LIN {X 0,Y 361.85,Z 263.036,A -85,B 0,C 180,E1 -12994.281,E2 -12994.281} C_VEL
LIN {X 0,Y 361.86,Z 263.015,A -85,B 0,C 180,E1 -12997.224,E2 -12997.224} C_VEL
LIN {X 0,Y 361.831,Z 263.036,A -85,B 0,C 180,E1 -13000.756,E2 -13000.756} C_VEL
LIN {X 0,Y 361.816,Z 263.041,A -85,B 0,C 180,E1 -13004.368,E2 -13004.368} C_VEL
LIN {X 0,Y 361.832,Z 262.994,A -85,B 0,C 180,E1 -13007.569,E2 -13007.569} C_VEL
LIN {X 0,Y 361.867,Z 263.034,A -85,B 0,C 180,E1 -13010.974,E2 -13010.974} C_VEL
LIN {X 0,Y 361.871,Z 263.004,A -85,B 0,C 180,E1 -13014.656,E2 -13014.656} C_VEL
LIN {X 0,Y 361.873,Z 263.221,A -85,B 0,C 180,E1 -13016.677,E2 -13016.677} C_VEL
LIN {X 0,Y 365.192,Z 275.83,A -85,B 0,C 180,E1 -13019.658,E2 -13019.658} C_VEL
LIN {X 0,Y 368.197,Z 288.508,A -85,B 0,C 180,E1 -13022.471,E2 -13022.471} C_VEL
LIN {X 0,Y 369.094,Z 293.338,A -85,B 0,C 180,E1 -13023.5,E2 -13023.5} C_VEL
LIN {X 0,Y 368.469,Z 298.908,A -85,B 0,C 180,E1 -13024.51,E2 -13024.51} C_VEL
LIN {X 0,Y 372.505,Z 325.5,A -85,B 0,C 180,E1 -13025.374,E2 -13025.374} C_VEL
LIN {X 0,Y 370.326,Z 430.343,A -85,B 0,C 180,E1 -13027.51,E2 -13027.51} C_VEL
LIN {X 0,Y 369.606,Z 444.397,A -85,B 0,C 180,E1 -13027.979,E2 -13027.979} C_VEL
LIN {X 0,Y 368.698,Z 458.571,A -85,B 0,C 180,E1 -13028.694,E2 -13028.694} C_VEL
LIN {X 0,Y 367.725,Z 471.328,A -85,B 0,C 180,E1 -13029.558,E2 -13029.558} C_VEL
LIN {X 0,Y 366.493,Z 484.339,A -85,B 0,C 180,E1 -13030.684,E2 -13030.684} C_VEL
LIN {X 0,Y 365.21,Z 495.855,A -85,B 0,C 180,E1 -13031.923,E2 -13031.923} C_VEL
LIN {X 0,Y 363.937,Z 507.367,A -85,B 0,C 180,E1 -13033.451,E2 -13033.451} C_VEL
LIN {X 0,Y 362.894,Z 517.59,A -85,B 0,C 180,E1 -13035.132,E2 -13035.132} C_VEL
LIN {X 0,Y 362.087,Z 526.041,A -85,B 0,C 180,E1 -13036.817,E2 -13036.817} C_VEL
LIN {X 0,Y 361.259,Z 534.081,A -85,B 0,C 180,E1 -13038.782,E2 -13038.782} C_VEL
LIN {X 0,Y 360.837,Z 539.679,A -85,B 0,C 180,E1 -13040.471,E2 -13040.471} C_VEL
LIN {X 0,Y 360.561,Z 544.242,A -85,B 0,C 180,E1 -13042.158,E2 -13042.158} C_VEL
LIN {X 0,Y 360.376,Z 548.192,A -85,B 0,C 180,E1 -13044.039,E2 -13044.039} C_VEL
LIN {X 0,Y 360.322,Z 550.495,A -85,B 0,C 180,E1 -13045.525,E2 -13045.525} C_VEL
LIN {X 0,Y 360.262,Z 552.787,A -85,B 0,C 180,E1 -13047.764,E2 -13047.764} C_VEL
LIN {X 0,Y 360.358,Z 553.65,A -85,B 0,C 180,E1 -13050,E2 -13050} C_VEL
LIN {X 0,Y 360.26,Z 553.086,A -85,B 0,C 180,E1 -13052.236,E2 -13052.236} C_VEL
LIN {X 0,Y 360.329,Z 551.079,A -85,B 0,C 180,E1 -13054.475,E2 -13054.475} C_VEL
LIN {X 0,Y 360.479,Z 547.581,A -85,B 0,C 180,E1 -13056.718,E2 -13056.718} C_VEL
LIN {X 0,Y 360.763,Z 542.513,A -85,B 0,C 180,E1 -13058.966,E2 -13058.966} C_VEL
LIN {X 0,Y 361.161,Z 537.589,A -85,B 0,C 180,E1 -13060.653,E2 -13060.653} C_VEL
LIN {X 0,Y 361.961,Z 530.449,A -85,B 0,C 180,E1 -13062.617,E2 -13062.617} C_VEL
LIN {X 0,Y 362.829,Z 522.364,A -85,B 0,C 180,E1 -13064.419,E2 -13064.419} C_VEL
LIN {X 0,Y 363.782,Z 513.901,A -85,B 0,C 180,E1 -13065.98,E2 -13065.98} C_VEL
LIN {X 0,Y 365.146,Z 502.912,A -85,B 0,C 180,E1 -13067.646,E2 -13067.646} C_VEL
LIN {X 0,Y 366.48,Z 491.723,A -85,B 0,C 180,E1 -13069.026,E2 -13069.026} C_VEL
LIN {X 0,Y 367.904,Z 479.321,A -85,B 0,C 180,E1 -13070.255,E2 -13070.255} C_VEL
LIN {X 0,Y 368.921,Z 468.55,A -85,B 0,C 180,E1 -13071.126,E2 -13071.126} C_VEL
LIN {X 0,Y 370.017,Z 455.357,A -85,B 0,C 180,E1 -13071.958,E2 -13071.958} C_VEL
LIN {X 0,Y 370.863,Z 442.406,A -85,B 0,C 180,E1 -13072.566,E2 -13072.566} C_VEL
LIN {X 0,Y 371.556,Z 428.554,A -85,B 0,C 180,E1 -13072.999,E2 -13072.999} C_VEL
LIN {X 0,Y 373.814,Z 326.139,A -85,B 0,C 180,E1 -13075.086,E2 -13075.086} C_VEL
LIN {X 0,Y 369.32,Z 299.055,A -85,B 0,C 180,E1 -13076.023,E2 -13076.023} C_VEL
LIN {X 0,Y 369.764,Z 294.707,A -85,B 0,C 180,E1 -13076.812,E2 -13076.812} C_VEL
LIN {X 0,Y 367.763,Z 285.49,A -85,B 0,C 180,E1 -13078.85,E2 -13078.85} C_VEL
LIN {X 0,Y 364.404,Z 272.229,A -85,B 0,C 180,E1 -13081.941,E2 -13081.941} C_VEL
LIN {X 0,Y 361.899,Z 263.126,A -85,B 0,C 180,E1 -13084.246,E2 -13084.246} C_VEL
LIN {X 0,Y 361.861,Z 263.004,A -85,B 0,C 180,E1 -13087.222,E2 -13087.222} C_VEL
LIN {X 0,Y 361.902,Z 263.021,A -85,B 0,C 180,E1 -13090.768,E2 -13090.768} C_VEL
LIN {X 0,Y 361.908,Z 263.017,A -85,B 0,C 180,E1 -13094.353,E2 -13094.353} C_VEL
LIN {X 0,Y 361.833,Z 263.032,A -85,B 0,C 180,E1 -13097.568,E2 -13097.568} C_VEL
LIN {X 0,Y 361.867,Z 263.034,A -85,B 0,C 180,E1 -13100.973,E2 -13100.973} C_VEL
LIN {X 0,Y 361.87,Z 263.017,A -85,B 0,C 180,E1 -13104.655,E2 -13104.655} C_VEL
LIN {X 0,Y 361.833,Z 263.029,A -85,B 0,C 180,E1 -13108.37,E2 -13108.37} C_VEL
LIN {X 0,Y 361.897,Z 263.009,A -85,B 0,C 180,E1 -13110.955,E2 -13110.955} C_VEL
LIN {X 0,Y 361.95,Z 263.023,A -85,B 0,C 180,E1 -13113.475,E2 -13113.475} C_VEL
LIN {X 0,Y 361.885,Z 263.03,A -85,B 0,C 180,E1 -13117.145,E2 -13117.145} C_VEL
LIN {X 0,Y 361.915,Z 263.026,A -85,B 0,C 180,E1 -13120.724,E2 -13120.724} C_VEL
LIN {X 0,Y 361.94,Z 263.019,A -85,B 0,C 180,E1 -13124.226,E2 -13124.226} C_VEL
LIN {X 0,Y 361.993,Z 263.015,A -85,B 0,C 180,E1 -13126.528,E2 -13126.528} C_VEL
LIN {X 0,Y 362.025,Z 263.016,A -85,B 0,C 180,E1 -13129.938,E2 -13129.938} C_VEL
LIN {X 0,Y 362.157,Z 262.988,A -85,B 0,C 180,E1 -13133.314,E2 -13133.314} C_VEL
LIN {X 0,Y 362.277,Z 262.975,A -85,B 0,C 180,E1 -13137.777,E2 -13137.777} C_VEL
LIN {X 0,Y 362.422,Z 262.965,A -85,B 0,C 180,E1 -13140,E2 -13140} C_VEL
LIN {X 0,Y 362.277,Z 262.972,A -85,B 0,C 180,E1 -13142.224,E2 -13142.224} C_VEL
LIN {X 0,Y 362.166,Z 262.989,A -85,B 0,C 180,E1 -13146.687,E2 -13146.687} C_VEL
LIN {X 0,Y 362.069,Z 263.007,A -85,B 0,C 180,E1 -13148.934,E2 -13148.934} C_VEL
LIN {X 0,Y 361.955,Z 263.017,A -85,B 0,C 180,E1 -13152.333,E2 -13152.333} C_VEL
LIN {X 0,Y 361.957,Z 263.021,A -85,B 0,C 180,E1 -13154.621,E2 -13154.621} C_VEL
LIN {X 0,Y 361.952,Z 263.022,A -85,B 0,C 180,E1 -13158.1,E2 -13158.1} C_VEL
LIN {X 0,Y 361.89,Z 263.032,A -85,B 0,C 180,E1 -13161.654,E2 -13161.654} C_VEL
LIN {X 0,Y 361.925,Z 263.03,A -85,B 0,C 180,E1 -13165.291,E2 -13165.291} C_VEL
LIN {X 0,Y 361.905,Z 263.016,A -85,B 0,C 180,E1 -13167.78,E2 -13167.78} C_VEL
LIN {X 0,Y 361.835,Z 263.039,A -85,B 0,C 180,E1 -13171.63,E2 -13171.63} C_VEL
LIN {X 0,Y 361.873,Z 263.016,A -85,B 0,C 180,E1 -13175.346,E2 -13175.346} C_VEL
LIN {X 0,Y 361.868,Z 263.023,A -85,B 0,C 180,E1 -13179.027,E2 -13179.027} C_VEL
LIN {X 0,Y 361.835,Z 263.035,A -85,B 0,C 180,E1 -13182.83,E2 -13182.83} C_VEL
LIN {X 0,Y 361.82,Z 263.042,A -85,B 0,C 180,E1 -13185.947,E2 -13185.947} C_VEL
LIN {X 0,Y 361.838,Z 263.039,A -85,B 0,C 180,E1 -13189.245,E2 -13189.245} C_VEL
LIN {X 0,Y 361.865,Z 263.007,A -85,B 0,C 180,E1 -13192.778,E2 -13192.778} C_VEL
LIN {X 0,Y 361.888,Z 263.182,A -85,B 0,C 180,E1 -13193.42,E2 -13193.42} C_VEL
LIN {X 0,Y 364.744,Z 273.91,A -85,B 0,C 180,E1 -13196.286,E2 -13196.286} C_VEL
LIN {X 0,Y 367.578,Z 286.235,A -85,B 0,C 180,E1 -13199.361,E2 -13199.361} C_VEL
LIN {X 0,Y 368.84,Z 292.603,A -85,B 0,C 180,E1 -13200.881,E2 -13200.881} C_VEL
LIN {X 0,Y 367.561,Z 304.193,A -85,B 0,C 180,E1 -13203.299,E2 -13203.299} C_VEL
LIN {X 0,Y 366.772,Z 311.792,A -85,B 0,C 180,E1 -13204.83,E2 -13204.83} C_VEL
LIN {X 0,Y 370.593,Z 331.748,A -85,B 0,C 180,E1 -13205.546,E2 -13205.546} C_VEL
LIN {X 0,Y 372.973,Z 345.776,A -85,B 0,C 180,E1 -13205.987,E2 -13205.987} C_VEL
LIN {X 0,Y 371.541,Z 426.495,A -85,B 0,C 180,E1 -13207.478,E2 -13207.478} C_VEL
LIN {X 0,Y 370.858,Z 439.638,A -85,B 0,C 180,E1 -13207.925,E2 -13207.925} C_VEL
LIN {X 0,Y 370.174,Z 451.942,A -85,B 0,C 180,E1 -13208.566,E2 -13208.566} C_VEL
LIN {X 0,Y 369.128,Z 463.623,A -85,B 0,C 180,E1 -13209.377,E2 -13209.377} C_VEL
LIN {X 0,Y 368.017,Z 474.31,A -85,B 0,C 180,E1 -13210.331,E2 -13210.331} C_VEL
LIN {X 0,Y 366.588,Z 485.271,A -85,B 0,C 180,E1 -13211.559,E2 -13211.559} C_VEL
LIN {X 0,Y 365.289,Z 495.077,A -85,B 0,C 180,E1 -13212.938,E2 -13212.938} C_VEL
LIN {X 0,Y 363.91,Z 504.604,A -85,B 0,C 180,E1 -13214.601,E2 -13214.601} C_VEL
LIN {X 0,Y 362.944,Z 512.259,A -85,B 0,C 180,E1 -13216.278,E2 -13216.278} C_VEL
LIN {X 0,Y 362.184,Z 517.473,A -85,B 0,C 180,E1 -13217.676,E2 -13217.676} C_VEL
LIN {X 0,Y 361.451,Z 522.599,A -85,B 0,C 180,E1 -13219.356,E2 -13219.356} C_VEL
LIN {X 0,Y 361.01,Z 526.617,A -85,B 0,C 180,E1 -13221.04,E2 -13221.04} C_VEL
LIN {X 0,Y 360.773,Z 528.765,A -85,B 0,C 180,E1 -13222.163,E2 -13222.163} C_VEL
LIN {X 0,Y 360.453,Z 531.766,A -85,B 0,C 180,E1 -13224.405,E2 -13224.405} C_VEL
LIN {X 0,Y 360.434,Z 532.696,A -85,B 0,C 180,E1 -13225.527,E2 -13225.527} C_VEL
LIN {X 0,Y 360.314,Z 533.479,A -85,B 0,C 180,E1 -13227.764,E2 -13227.764} C_VEL
LIN {X 0,Y 360.365,Z 532.757,A -85,B 0,C 180,E1 -13230,E2 -13230} C_VEL
LIN {X 0,Y 360.523,Z 530.577,A -85,B 0,C 180,E1 -13232.234,E2 -13232.234} C_VEL
LIN {X 0,Y 360.806,Z 527.911,A -85,B 0,C 180,E1 -13233.909,E2 -13233.909} C_VEL
LIN {X 0,Y 361.087,Z 524.308,A -85,B 0,C 180,E1 -13235.585,E2 -13235.585} C_VEL
LIN {X 0,Y 361.638,Z 519.475,A -85,B 0,C 180,E1 -13237.314,E2 -13237.314} C_VEL
LIN {X 0,Y 362.399,Z 512.737,A -85,B 0,C 180,E1 -13239.206,E2 -13239.206} C_VEL
LIN {X 0,Y 363.371,Z 505.272,A -85,B 0,C 180,E1 -13240.869,E2 -13240.869} C_VEL
LIN {X 0,Y 364.513,Z 495.956,A -85,B 0,C 180,E1 -13242.527,E2 -13242.527} C_VEL
LIN {X 0,Y 365.736,Z 485.342,A -85,B 0,C 180,E1 -13244.04,E2 -13244.04} C_VEL
LIN {X 0,Y 366.995,Z 474.475,A -85,B 0,C 180,E1 -13245.266,E2 -13245.266} C_VEL
LIN {X 0,Y 368.083,Z 463.896,A -85,B 0,C 180,E1 -13246.215,E2 -13246.215} C_VEL
LIN {X 0,Y 368.993,Z 452.347,A -85,B 0,C 180,E1 -13247.028,E2 -13247.028} C_VEL
LIN {X 0,Y 369.639,Z 442.84,A -85,B 0,C 180,E1 -13247.543,E2 -13247.543} C_VEL
LIN {X 0,Y 369.41,Z 437.209,A -85,B 0,C 180,E1 -13247.819,E2 -13247.819} C_VEL
LIN {X 0,Y 367.06,Z 428.039,A -85,B 0,C 180,E1 -13248.284,E2 -13248.284} C_VEL
LIN {X 0,Y 364.522,Z 418.753,A -85,B 0,C 180,E1 -13248.664,E2 -13248.664} C_VEL
LIN {X 0,Y 364.025,Z 412.941,A -85,B 0,C 180,E1 -13248.805,E2 -13248.805} C_VEL
LIN {X 0,Y 364.996,Z 345.148,A -85,B 0,C 180,E1 -13250.065,E2 -13250.065} C_VEL
LIN {X 0,Y 359.954,Z 315.672,A -85,B 0,C 180,E1 -13250.989,E2 -13250.989} C_VEL
LIN {X 0,Y 359.295,Z 311.586,A -85,B 0,C 180,E1 -13251.172,E2 -13251.172} C_VEL
LIN {X 0,Y 361.123,Z 294.445,A -85,B 0,C 180,E1 -13254.734,E2 -13254.734} C_VEL
LIN {X 0,Y 361.222,Z 291.662,A -85,B 0,C 180,E1 -13255.342,E2 -13255.342} C_VEL
LIN {X 0,Y 358.66,Z 279.164,A -85,B 0,C 180,E1 -13258.37,E2 -13258.37} C_VEL
LIN {X 0,Y 355.383,Z 266.058,A -85,B 0,C 180,E1 -13261.748,E2 -13261.748} C_VEL
LIN {X 0,Y 354.827,Z 263.972,A -85,B 0,C 180,E1 -13262.371,E2 -13262.371} C_VEL
LIN {X 0,Y 354.823,Z 263.909,A -85,B 0,C 180,E1 -13265.698,E2 -13265.698} C_VEL
LIN {X 0,Y 354.824,Z 263.913,A -85,B 0,C 180,E1 -13269.423,E2 -13269.423} C_VEL
LIN {X 0,Y 354.788,Z 263.917,A -85,B 0,C 180,E1 -13272.866,E2 -13272.866} C_VEL
LIN {X 0,Y 354.766,Z 263.911,A -85,B 0,C 180,E1 -13276.103,E2 -13276.103} C_VEL
LIN {X 0,Y 354.786,Z 263.901,A -85,B 0,C 180,E1 -13279.178,E2 -13279.178} C_VEL
LIN {X 0,Y 354.805,Z 263.911,A -85,B 0,C 180,E1 -13282.402,E2 -13282.402} C_VEL
LIN {X 0,Y 354.809,Z 263.897,A -85,B 0,C 180,E1 -13284.94,E2 -13284.94} C_VEL
LIN {X 0,Y 354.791,Z 263.908,A -85,B 0,C 180,E1 -13288.404,E2 -13288.404} C_VEL
LIN {X 0,Y 354.851,Z 263.9,A -85,B 0,C 180,E1 -13291.618,E2 -13291.618} C_VEL
LIN {X 0,Y 354.895,Z 263.902,A -85,B 0,C 180,E1 -13294.172,E2 -13294.172} C_VEL
LIN {X 0,Y 354.828,Z 263.909,A -85,B 0,C 180,E1 -13297.893,E2 -13297.893} C_VEL
LIN {X 0,Y 354.918,Z 263.897,A -85,B 0,C 180,E1 -13301.891,E2 -13301.891} C_VEL
LIN {X 0,Y 354.937,Z 263.89,A -85,B 0,C 180,E1 -13305.981,E2 -13305.981} C_VEL
LIN {X 0,Y 354.972,Z 263.884,A -85,B 0,C 180,E1 -13309.735,E2 -13309.735} C_VEL
LIN {X 0,Y 355.12,Z 263.873,A -85,B 0,C 180,E1 -13313.18,E2 -13313.18} C_VEL
LIN {X 0,Y 355.24,Z 263.858,A -85,B 0,C 180,E1 -13317.732,E2 -13317.732} C_VEL
LIN {X 0,Y 355.391,Z 263.834,A -85,B 0,C 180,E1 -13320,E2 -13320} C_VEL
LIN {X 0,Y 355.24,Z 263.856,A -85,B 0,C 180,E1 -13322.267,E2 -13322.267} C_VEL
LIN {X 0,Y 355.131,Z 263.868,A -85,B 0,C 180,E1 -13326.819,E2 -13326.819} C_VEL
LIN {X 0,Y 355.009,Z 263.885,A -85,B 0,C 180,E1 -13329.112,E2 -13329.112} C_VEL
LIN {X 0,Y 354.914,Z 263.9,A -85,B 0,C 180,E1 -13332.581,E2 -13332.581} C_VEL
LIN {X 0,Y 354.883,Z 263.896,A -85,B 0,C 180,E1 -13336.096,E2 -13336.096} C_VEL
LIN {X 0,Y 354.897,Z 263.903,A -85,B 0,C 180,E1 -13338.472,E2 -13338.472} C_VEL
LIN {X 0,Y 354.829,Z 263.911,A -85,B 0,C 180,E1 -13342.106,E2 -13342.106} C_VEL
LIN {X 0,Y 354.894,Z 263.899,A -85,B 0,C 180,E1 -13345.828,E2 -13345.828} C_VEL
LIN {X 0,Y 354.849,Z 263.885,A -85,B 0,C 180,E1 -13349.679,E2 -13349.679} C_VEL
LIN {X 0,Y 354.801,Z 263.916,A -85,B 0,C 180,E1 -13353.702,E2 -13353.702} C_VEL
LIN {X 0,Y 354.793,Z 263.895,A -85,B 0,C 180,E1 -13356.46,E2 -13356.46} C_VEL
LIN {X 0,Y 354.819,Z 263.914,A -85,B 0,C 180,E1 -13359.424,E2 -13359.424} C_VEL
LIN {X 0,Y 354.784,Z 263.906,A -85,B 0,C 180,E1 -13362.868,E2 -13362.868} C_VEL
LIN {X 0,Y 354.777,Z 263.898,A -85,B 0,C 180,E1 -13366.106,E2 -13366.106} C_VEL
LIN {X 0,Y 354.783,Z 263.875,A -85,B 0,C 180,E1 -13369.179,E2 -13369.179} C_VEL
LIN {X 0,Y 354.804,Z 263.902,A -85,B 0,C 180,E1 -13372.403,E2 -13372.403} C_VEL
LIN {X 0,Y 354.818,Z 263.969,A -85,B 0,C 180,E1 -13376.07,E2 -13376.07} C_VEL
LIN {X 0,Y 357.55,Z 274.162,A -85,B 0,C 180,E1 -13378.609,E2 -13378.609} C_VEL
LIN {X 0,Y 360.996,Z 288.429,A -85,B 0,C 180,E1 -13381.885,E2 -13381.885} C_VEL
LIN {X 0,Y 362.224,Z 294.363,A -85,B 0,C 180,E1 -13383.19,E2 -13383.19} C_VEL
LIN {X 0,Y 361.79,Z 299.207,A -85,B 0,C 180,E1 -13384.068,E2 -13384.068} C_VEL
LIN {X 0,Y 365.954,Z 326.74,A -85,B 0,C 180,E1 -13384.977,E2 -13384.977} C_VEL
LIN {X 0,Y 363.665,Z 431.378,A -85,B 0,C 180,E1 -13387.15,E2 -13387.15} C_VEL
LIN {X 0,Y 362.85,Z 445.727,A -85,B 0,C 180,E1 -13387.66,E2 -13387.66} C_VEL
LIN {X 0,Y 361.875,Z 459.999,A -85,B 0,C 180,E1 -13388.414,E2 -13388.414} C_VEL
LIN {X 0,Y 360.84,Z 473.26,A -85,B 0,C 180,E1 -13389.361,E2 -13389.361} C_VEL
LIN {X 0,Y 359.604,Z 485.281,A -85,B 0,C 180,E1 -13390.447,E2 -13390.447} C_VEL
LIN {X 0,Y 358.266,Z 496.607,A -85,B 0,C 180,E1 -13391.708,E2 -13391.708} C_VEL
LIN {X 0,Y 357.079,Z 506.996,A -85,B 0,C 180,E1 -13393.124,E2 -13393.124} C_VEL
LIN {X 0,Y 355.968,Z 517.258,A -85,B 0,C 180,E1 -13394.835,E2 -13394.835} C_VEL
LIN {X 0,Y 355.143,Z 525.738,A -85,B 0,C 180,E1 -13396.555,E2 -13396.555} C_VEL
LIN {X 0,Y 354.265,Z 533.801,A -85,B 0,C 180,E1 -13398.558,E2 -13398.558} C_VEL
LIN {X 0,Y 353.787,Z 539.417,A -85,B 0,C 180,E1 -13400.279,E2 -13400.279} C_VEL
LIN {X 0,Y 353.492,Z 543.998,A -85,B 0,C 180,E1 -13402,E2 -13402} C_VEL
LIN {X 0,Y 353.276,Z 548.246,A -85,B 0,C 180,E1 -13404.092,E2 -13404.092} C_VEL
LIN {X 0,Y 353.235,Z 550.272,A -85,B 0,C 180,E1 -13405.435,E2 -13405.435} C_VEL
LIN {X 0,Y 353.17,Z 552.576,A -85,B 0,C 180,E1 -13407.719,E2 -13407.719} C_VEL
LIN {X 0,Y 353.26,Z 553.448,A -85,B 0,C 180,E1 -13410,E2 -13410} C_VEL
LIN {X 0,Y 353.168,Z 552.894,A -85,B 0,C 180,E1 -13412.281,E2 -13412.281} C_VEL
LIN {X 0,Y 353.243,Z 550.899,A -85,B 0,C 180,E1 -13414.565,E2 -13414.565} C_VEL
LIN {X 0,Y 353.388,Z 547.406,A -85,B 0,C 180,E1 -13416.853,E2 -13416.853} C_VEL
LIN {X 0,Y 353.701,Z 542.345,A -85,B 0,C 180,E1 -13419.146,E2 -13419.146} C_VEL
LIN {X 0,Y 354.126,Z 537.425,A -85,B 0,C 180,E1 -13420.867,E2 -13420.867} C_VEL
LIN {X 0,Y 354.983,Z 530.289,A -85,B 0,C 180,E1 -13422.869,E2 -13422.869} C_VEL
LIN {X 0,Y 356.013,Z 521.414,A -85,B 0,C 180,E1 -13424.87,E2 -13424.87} C_VEL
LIN {X 0,Y 357.153,Z 512.096,A -85,B 0,C 180,E1 -13426.578,E2 -13426.578} C_VEL
LIN {X 0,Y 358.481,Z 501.752,A -85,B 0,C 180,E1 -13428.133,E2 -13428.133} C_VEL
LIN {X 0,Y 359.937,Z 490.281,A -85,B 0,C 180,E1 -13429.534,E2 -13429.534} C_VEL
LIN {X 0,Y 361.329,Z 477.518,A -85,B 0,C 180,E1 -13430.794,E2 -13430.794} C_VEL
LIN {X 0,Y 362.584,Z 465.109,A -85,B 0,C 180,E1 -13431.759,E2 -13431.759} C_VEL
LIN {X 0,Y 363.69,Z 451.275,A -85,B 0,C 180,E1 -13432.585,E2 -13432.585} C_VEL
LIN {X 0,Y 364.624,Z 437.641,A -85,B 0,C 180,E1 -13433.161,E2 -13433.161} C_VEL
LIN {X 0,Y 365.152,Z 423.665,A -85,B 0,C 180,E1 -13433.538,E2 -13433.538} C_VEL
LIN {X 0,Y 367.31,Z 326.411,A -85,B 0,C 180,E1 -13435.545,E2 -13435.545} C_VEL
LIN {X 0,Y 362.731,Z 299.025,A -85,B 0,C 180,E1 -13436.535,E2 -13436.535} C_VEL
LIN {X 0,Y 362.956,Z 296.33,A -85,B 0,C 180,E1 -13437.038,E2 -13437.038} C_VEL
LIN {X 0,Y 360.625,Z 285.59,A -85,B 0,C 180,E1 -13439.477,E2 -13439.477} C_VEL
LIN {X 0,Y 357.059,Z 271.925,A -85,B 0,C 180,E1 -13442.77,E2 -13442.77} C_VEL
LIN {X 0,Y 354.844,Z 263.997,A -85,B 0,C 180,E1 -13444.848,E2 -13444.848} C_VEL
LIN {X 0,Y 354.803,Z 263.892,A -85,B 0,C 180,E1 -13447.882,E2 -13447.882} C_VEL
LIN {X 0,Y 354.835,Z 263.901,A -85,B 0,C 180,E1 -13451.18,E2 -13451.18} C_VEL
LIN {X 0,Y 354.859,Z 263.895,A -85,B 0,C 180,E1 -13454.522,E2 -13454.522} C_VEL
LIN {X 0,Y 354.791,Z 263.907,A -85,B 0,C 180,E1 -13457.662,E2 -13457.662} C_VEL
LIN {X 0,Y 354.811,Z 263.914,A -85,B 0,C 180,E1 -13460.666,E2 -13460.666} C_VEL
LIN {X 0,Y 354.818,Z 263.892,A -85,B 0,C 180,E1 -13464.3,E2 -13464.3} C_VEL
LIN {X 0,Y 354.782,Z 263.916,A -85,B 0,C 180,E1 -13467.666,E2 -13467.666} C_VEL
LIN {X 0,Y 354.864,Z 263.881,A -85,B 0,C 180,E1 -13470.621,E2 -13470.621} C_VEL
LIN {X 0,Y 354.894,Z 263.902,A -85,B 0,C 180,E1 -13474.172,E2 -13474.172} C_VEL
LIN {X 0,Y 354.829,Z 263.912,A -85,B 0,C 180,E1 -13477.894,E2 -13477.894} C_VEL
LIN {X 0,Y 354.918,Z 263.901,A -85,B 0,C 180,E1 -13481.891,E2 -13481.891} C_VEL
LIN {X 0,Y 354.937,Z 263.898,A -85,B 0,C 180,E1 -13485.981,E2 -13485.981} C_VEL
LIN {X 0,Y 354.972,Z 263.892,A -85,B 0,C 180,E1 -13489.736,E2 -13489.736} C_VEL
LIN {X 0,Y 355.121,Z 263.863,A -85,B 0,C 180,E1 -13493.181,E2 -13493.181} C_VEL
LIN {X 0,Y 355.24,Z 263.851,A -85,B 0,C 180,E1 -13497.733,E2 -13497.733} C_VEL
LIN {X 0,Y 355.392,Z 263.84,A -85,B 0,C 180,E1 -13500,E2 -13500} C_VEL
LIN {X 0,Y 355.24,Z 263.849,A -85,B 0,C 180,E1 -13502.268,E2 -13502.268} C_VEL
LIN {X 0,Y 355.133,Z 263.864,A -85,B 0,C 180,E1 -13506.82,E2 -13506.82} C_VEL
LIN {X 0,Y 355.01,Z 263.888,A -85,B 0,C 180,E1 -13509.113,E2 -13509.113} C_VEL
LIN {X 0,Y 354.916,Z 263.894,A -85,B 0,C 180,E1 -13512.582,E2 -13512.582} C_VEL
LIN {X 0,Y 354.885,Z 263.896,A -85,B 0,C 180,E1 -13516.097,E2 -13516.097} C_VEL
LIN {X 0,Y 354.897,Z 263.901,A -85,B 0,C 180,E1 -13518.473,E2 -13518.473} C_VEL
LIN {X 0,Y 354.832,Z 263.909,A -85,B 0,C 180,E1 -13522.107,E2 -13522.107} C_VEL
LIN {X 0,Y 354.896,Z 263.902,A -85,B 0,C 180,E1 -13525.828,E2 -13525.828} C_VEL
LIN {X 0,Y 354.815,Z 263.891,A -85,B 0,C 180,E1 -13529.683,E2 -13529.683} C_VEL
LIN {X 0,Y 354.804,Z 263.906,A -85,B 0,C 180,E1 -13533.703,E2 -13533.703} C_VEL
LIN {X 0,Y 354.799,Z 263.906,A -85,B 0,C 180,E1 -13536.46,E2 -13536.46} C_VEL
LIN {X 0,Y 354.823,Z 263.897,A -85,B 0,C 180,E1 -13539.425,E2 -13539.425} C_VEL
LIN {X 0,Y 354.787,Z 263.913,A -85,B 0,C 180,E1 -13542.868,E2 -13542.868} C_VEL
LIN {X 0,Y 354.769,Z 263.921,A -85,B 0,C 180,E1 -13546.105,E2 -13546.105} C_VEL
LIN {X 0,Y 354.79,Z 263.918,A -85,B 0,C 180,E1 -13549.18,E2 -13549.18} C_VEL
LIN {X 0,Y 354.844,Z 264.023,A -85,B 0,C 180,E1 -13552.811,E2 -13552.811} C_VEL
LIN {X 0,Y 357.595,Z 274.245,A -85,B 0,C 180,E1 -13555.635,E2 -13555.635} C_VEL
LIN {X 0,Y 360.671,Z 287.482,A -85,B 0,C 180,E1 -13559.025,E2 -13559.025} C_VEL
LIN {X 0,Y 362.001,Z 294.128,A -85,B 0,C 180,E1 -13560.647,E2 -13560.647} C_VEL
LIN {X 0,Y 361.283,Z 301.246,A -85,B 0,C 180,E1 -13562.169,E2 -13562.169} C_VEL
LIN {X 0,Y 360.095,Z 311.644,A -85,B 0,C 180,E1 -13564.32,E2 -13564.32} C_VEL
LIN {X 0,Y 364.167,Z 332.827,A -85,B 0,C 180,E1 -13565.102,E2 -13565.102} C_VEL
LIN {X 0,Y 366.514,Z 346.606,A -85,B 0,C 180,E1 -13565.548,E2 -13565.548} C_VEL
LIN {X 0,Y 365.011,Z 426.627,A -85,B 0,C 180,E1 -13567.052,E2 -13567.052} C_VEL
LIN {X 0,Y 364.271,Z 439.964,A -85,B 0,C 180,E1 -13567.515,E2 -13567.515} C_VEL
LIN {X 0,Y 363.57,Z 452.04,A -85,B 0,C 180,E1 -13568.157,E2 -13568.157} C_VEL
LIN {X 0,Y 362.495,Z 463.721,A -85,B 0,C 180,E1 -13568.981,E2 -13568.981} C_VEL
LIN {X 0,Y 361.326,Z 474.411,A -85,B 0,C 180,E1 -13569.952,E2 -13569.952} C_VEL
LIN {X 0,Y 359.861,Z 485.379,A -85,B 0,C 180,E1 -13571.202,E2 -13571.202} C_VEL
LIN {X 0,Y 358.474,Z 495.191,A -85,B 0,C 180,E1 -13572.604,E2 -13572.604} C_VEL
LIN {X 0,Y 357.046,Z 504.726,A -85,B 0,C 180,E1 -13574.298,E2 -13574.298} C_VEL
LIN {X 0,Y 356,Z 512.427,A -85,B 0,C 180,E1 -13576.014,E2 -13576.014} C_VEL
LIN {X 0,Y 355.245,Z 517.612,A -85,B 0,C 180,E1 -13577.431,E2 -13577.431} C_VEL
LIN {X 0,Y 354.451,Z 522.747,A -85,B 0,C 180,E1 -13579.143,E2 -13579.143} C_VEL
LIN {X 0,Y 353.96,Z 526.776,A -85,B 0,C 180,E1 -13580.86,E2 -13580.86} C_VEL
LIN {X 0,Y 353.719,Z 528.928,A -85,B 0,C 180,E1 -13582.005,E2 -13582.005} C_VEL
LIN {X 0,Y 353.438,Z 531.496,A -85,B 0,C 180,E1 -13583.851,E2 -13583.851} C_VEL
LIN {X 0,Y 353.344,Z 532.88,A -85,B 0,C 180,E1 -13585.437,E2 -13585.437} C_VEL
LIN {X 0,Y 353.22,Z 533.675,A -85,B 0,C 180,E1 -13587.719,E2 -13587.719} C_VEL
LIN {X 0,Y 353.247,Z 533.512,A -85,B 0,C 180,E1 -13588.86,E2 -13588.86} C_VEL
LIN {X 0,Y 353.323,Z 532.073,A -85,B 0,C 180,E1 -13591.14,E2 -13591.14} C_VEL
LIN {X 0,Y 353.588,Z 529.163,A -85,B 0,C 180,E1 -13593.418,E2 -13593.418} C_VEL
LIN {X 0,Y 353.882,Z 525.888,A -85,B 0,C 180,E1 -13595.127,E2 -13595.127} C_VEL
LIN {X 0,Y 354.413,Z 521.609,A -85,B 0,C 180,E1 -13596.833,E2 -13596.833} C_VEL
LIN {X 0,Y 355.141,Z 515.218,A -85,B 0,C 180,E1 -13598.822,E2 -13598.822} C_VEL
LIN {X 0,Y 356.011,Z 508.264,A -85,B 0,C 180,E1 -13600.521,E2 -13600.521} C_VEL
LIN {X 0,Y 357.204,Z 499.651,A -85,B 0,C 180,E1 -13602.21,E2 -13602.21} C_VEL
LIN {X 0,Y 358.315,Z 490.874,A -85,B 0,C 180,E1 -13603.613,E2 -13603.613} C_VEL
LIN {X 0,Y 359.457,Z 481.27,A -85,B 0,C 180,E1 -13604.869,E2 -13604.869} C_VEL
LIN {X 0,Y 360.584,Z 470.793,A -85,B 0,C 180,E1 -13605.98,E2 -13605.98} C_VEL
LIN {X 0,Y 361.73,Z 459.246,A -85,B 0,C 180,E1 -13606.943,E2 -13606.943} C_VEL
LIN {X 0,Y 362.688,Z 447.317,A -85,B 0,C 180,E1 -13607.697,E2 -13607.697} C_VEL
LIN {X 0,Y 363.383,Z 434.196,A -85,B 0,C 180,E1 -13608.29,E2 -13608.29} C_VEL
LIN {X 0,Y 363.859,Z 420.763,A -85,B 0,C 180,E1 -13608.662,E2 -13608.662} C_VEL
LIN {X 0,Y 364.025,Z 412.941,A -85,B 0,C 180,E1 -13608.805,E2 -13608.805} C_VEL
LIN {X 0,Y 363.616,Z 407.128,A -85,B 0,C 180,E1 -13608.943,E2 -13608.943} C_VEL
LIN {X 0,Y 359.05,Z 390.31,A -85,B 0,C 180,E1 -13609.561,E2 -13609.561} C_VEL
LIN {X 0,Y 358.046,Z 384.566,A -85,B 0,C 180,E1 -13609.74,E2 -13609.74} C_VEL
LIN {X 0,Y 357.93,Z 382.612,A -85,B 0,C 180,E1 -13609.787,E2 -13609.787} C_VEL
LIN {X 0,Y 358.472,Z 346.101,A -85,B 0,C 180,E1 -13610.479,E2 -13610.479} C_VEL
LIN {X 0,Y 352.932,Z 313.976,A -85,B 0,C 180,E1 -13611.52,E2 -13611.52} C_VEL
LIN {X 0,Y 352.566,Z 311.323,A -85,B 0,C 180,E1 -13611.673,E2 -13611.673} C_VEL
LIN {X 0,Y 354.482,Z 294.556,A -85,B 0,C 180,E1 -13615.23,E2 -13615.23} C_VEL
LIN {X 0,Y 352.44,Z 283.633,A -85,B 0,C 180,E1 -13617.9,E2 -13617.9} C_VEL
LIN {X 0,Y 349.685,Z 272.324,A -85,B 0,C 180,E1 -13620.829,E2 -13620.829} C_VEL
LIN {X 0,Y 347.779,Z 264.846,A -85,B 0,C 180,E1 -13622.922,E2 -13622.922} C_VEL
LIN {X 0,Y 347.771,Z 264.794,A -85,B 0,C 180,E1 -13626.064,E2 -13626.064} C_VEL
LIN {X 0,Y 347.753,Z 264.791,A -85,B 0,C 180,E1 -13628.792,E2 -13628.792} C_VEL
LIN {X 0,Y 347.751,Z 264.786,A -85,B 0,C 180,E1 -13631.829,E2 -13631.829} C_VEL
LIN {X 0,Y 347.705,Z 264.784,A -85,B 0,C 180,E1 -13635.026,E2 -13635.026} C_VEL
LIN {X 0,Y 347.749,Z 264.791,A -85,B 0,C 180,E1 -13638.396,E2 -13638.396} C_VEL
LIN {X 0,Y 347.772,Z 264.787,A -85,B 0,C 180,E1 -13642.01,E2 -13642.01} C_VEL
LIN {X 0,Y 347.742,Z 264.77,A -85,B 0,C 180,E1 -13645.535,E2 -13645.535} C_VEL
LIN {X 0,Y 347.761,Z 264.791,A -85,B 0,C 180,E1 -13649.653,E2 -13649.653} C_VEL
LIN {X 0,Y 347.849,Z 264.776,A -85,B 0,C 180,E1 -13652.744,E2 -13652.744} C_VEL
LIN {X 0,Y 347.782,Z 264.778,A -85,B 0,C 180,E1 -13656.161,E2 -13656.161} C_VEL
LIN {X 0,Y 347.808,Z 264.778,A -85,B 0,C 180,E1 -13659.909,E2 -13659.909} C_VEL
LIN {X 0,Y 347.861,Z 264.778,A -85,B 0,C 180,E1 -13662.359,E2 -13662.359} C_VEL
LIN {X 0,Y 347.893,Z 264.767,A -85,B 0,C 180,E1 -13665.97,E2 -13665.97} C_VEL
LIN {X 0,Y 347.923,Z 264.762,A -85,B 0,C 180,E1 -13669.525,E2 -13669.525} C_VEL
LIN {X 0,Y 348.086,Z 264.75,A -85,B 0,C 180,E1 -13673.042,E2 -13673.042} C_VEL
LIN {X 0,Y 348.202,Z 264.734,A -85,B 0,C 180,E1 -13677.686,E2 -13677.686} C_VEL
LIN {X 0,Y 348.34,Z 264.712,A -85,B 0,C 180,E1 -13680,E2 -13680} C_VEL
LIN {X 0,Y 348.202,Z 264.733,A -85,B 0,C 180,E1 -13682.313,E2 -13682.313} C_VEL
LIN {X 0,Y 348.1,Z 264.745,A -85,B 0,C 180,E1 -13686.957,E2 -13686.957} C_VEL
LIN {X 0,Y 347.961,Z 264.763,A -85,B 0,C 180,E1 -13689.298,E2 -13689.298} C_VEL
LIN {X 0,Y 347.883,Z 264.775,A -85,B 0,C 180,E1 -13692.839,E2 -13692.839} C_VEL
LIN {X 0,Y 347.833,Z 264.775,A -85,B 0,C 180,E1 -13696.431,E2 -13696.431} C_VEL
LIN {X 0,Y 347.847,Z 264.778,A -85,B 0,C 180,E1 -13698.86,E2 -13698.86} C_VEL
LIN {X 0,Y 347.768,Z 264.791,A -85,B 0,C 180,E1 -13702.579,E2 -13702.579} C_VEL
LIN {X 0,Y 347.806,Z 264.778,A -85,B 0,C 180,E1 -13705.109,E2 -13705.109} C_VEL
LIN {X 0,Y 347.807,Z 264.785,A -85,B 0,C 180,E1 -13707.694,E2 -13707.694} C_VEL
LIN {X 0,Y 347.759,Z 264.764,A -85,B 0,C 180,E1 -13710.347,E2 -13710.347} C_VEL
LIN {X 0,Y 347.74,Z 264.793,A -85,B 0,C 180,E1 -13714.464,E2 -13714.464} C_VEL
LIN {X 0,Y 347.77,Z 264.777,A -85,B 0,C 180,E1 -13717.989,E2 -13717.989} C_VEL
LIN {X 0,Y 347.746,Z 264.779,A -85,B 0,C 180,E1 -13721.831,E2 -13721.831} C_VEL
LIN {X 0,Y 347.762,Z 264.79,A -85,B 0,C 180,E1 -13725.017,E2 -13725.017} C_VEL
LIN {X 0,Y 347.746,Z 264.744,A -85,B 0,C 180,E1 -13728.398,E2 -13728.398} C_VEL
LIN {X 0,Y 347.771,Z 264.787,A -85,B 0,C 180,E1 -13732.012,E2 -13732.012} C_VEL
LIN {X 0,Y 347.83,Z 264.958,A -85,B 0,C 180,E1 -13735.578,E2 -13735.578} C_VEL
LIN {X 0,Y 351.057,Z 277.165,A -85,B 0,C 180,E1 -13738.634,E2 -13738.634} C_VEL
LIN {X 0,Y 354.39,Z 291.12,A -85,B 0,C 180,E1 -13741.902,E2 -13741.902} C_VEL
LIN {X 0,Y 355.396,Z 296.629,A -85,B 0,C 180,E1 -13743.126,E2 -13743.126} C_VEL
LIN {X 0,Y 355.127,Z 299.246,A -85,B 0,C 180,E1 -13743.593,E2 -13743.593} C_VEL
LIN {X 0,Y 359.412,Z 327.817,A -85,B 0,C 180,E1 -13744.561,E2 -13744.561} C_VEL
LIN {X 0,Y 357.057,Z 431.128,A -85,B 0,C 180,E1 -13746.741,E2 -13746.741} C_VEL
LIN {X 0,Y 356.231,Z 445.546,A -85,B 0,C 180,E1 -13747.26,E2 -13747.26} C_VEL
LIN {X 0,Y 355.243,Z 459.377,A -85,B 0,C 180,E1 -13747.997,E2 -13747.997} C_VEL
LIN {X 0,Y 354.139,Z 472.67,A -85,B 0,C 180,E1 -13748.953,E2 -13748.953} C_VEL
LIN {X 0,Y 352.903,Z 484.785,A -85,B 0,C 180,E1 -13750.06,E2 -13750.06} C_VEL
LIN {X 0,Y 351.466,Z 496.175,A -85,B 0,C 180,E1 -13751.341,E2 -13751.341} C_VEL
LIN {X 0,Y 350.232,Z 506.621,A -85,B 0,C 180,E1 -13752.784,E2 -13752.784} C_VEL
LIN {X 0,Y 349.04,Z 516.927,A -85,B 0,C 180,E1 -13754.527,E2 -13754.527} C_VEL
LIN {X 0,Y 348.198,Z 525.436,A -85,B 0,C 180,E1 -13756.281,E2 -13756.281} C_VEL
LIN {X 0,Y 347.281,Z 533.521,A -85,B 0,C 180,E1 -13758.325,E2 -13758.325} C_VEL
LIN {X 0,Y 346.726,Z 539.156,A -85,B 0,C 180,E1 -13760.079,E2 -13760.079} C_VEL
LIN {X 0,Y 346.418,Z 543.753,A -85,B 0,C 180,E1 -13761.836,E2 -13761.836} C_VEL
LIN {X 0,Y 346.232,Z 547.343,A -85,B 0,C 180,E1 -13763.59,E2 -13763.59} C_VEL
LIN {X 0,Y 346.132,Z 550.048,A -85,B 0,C 180,E1 -13765.342,E2 -13765.342} C_VEL
LIN {X 0,Y 346.132,Z 551.389,A -85,B 0,C 180,E1 -13766.508,E2 -13766.508} C_VEL
LIN {X 0,Y 346.114,Z 552.984,A -85,B 0,C 180,E1 -13768.837,E2 -13768.837} C_VEL
LIN {X 0,Y 346.163,Z 553.247,A -85,B 0,C 180,E1 -13770,E2 -13770} C_VEL
LIN {X 0,Y 346.079,Z 552.703,A -85,B 0,C 180,E1 -13772.328,E2 -13772.328} C_VEL
LIN {X 0,Y 346.132,Z 551.896,A -85,B 0,C 180,E1 -13773.492,E2 -13773.492} C_VEL
LIN {X 0,Y 346.199,Z 549.164,A -85,B 0,C 180,E1 -13775.826,E2 -13775.826} C_VEL
LIN {X 0,Y 346.431,Z 544.908,A -85,B 0,C 180,E1 -13778.164,E2 -13778.164} C_VEL
LIN {X 0,Y 346.94,Z 539.019,A -85,B 0,C 180,E1 -13780.504,E2 -13780.504} C_VEL
LIN {X 0,Y 347.743,Z 532.352,A -85,B 0,C 180,E1 -13782.548,E2 -13782.548} C_VEL
LIN {X 0,Y 348.737,Z 524.422,A -85,B 0,C 180,E1 -13784.5,E2 -13784.5} C_VEL
LIN {X 0,Y 349.835,Z 515.246,A -85,B 0,C 180,E1 -13786.335,E2 -13786.335} C_VEL
LIN {X 0,Y 351.297,Z 504.581,A -85,B 0,C 180,E1 -13788.064,E2 -13788.064} C_VEL
LIN {X 0,Y 352.7,Z 493.788,A -85,B 0,C 180,E1 -13789.497,E2 -13789.497} C_VEL
LIN {X 0,Y 354.225,Z 481.961,A -85,B 0,C 180,E1 -13790.772,E2 -13790.772} C_VEL
LIN {X 0,Y 355.485,Z 469.933,A -85,B 0,C 180,E1 -13791.818,E2 -13791.818} C_VEL
LIN {X 0,Y 356.656,Z 457.376,A -85,B 0,C 180,E1 -13792.673,E2 -13792.673} C_VEL
LIN {X 0,Y 357.687,Z 443.668,A -85,B 0,C 180,E1 -13793.369,E2 -13793.369} C_VEL
LIN {X 0,Y 358.461,Z 429.23,A -85,B 0,C 180,E1 -13793.852,E2 -13793.852} C_VEL
LIN {X 0,Y 360.898,Z 327.396,A -85,B 0,C 180,E1 -13795.999,E2 -13795.999} C_VEL
LIN {X 0,Y 356.189,Z 299.398,A -85,B 0,C 180,E1 -13797.024,E2 -13797.024} C_VEL
LIN {X 0,Y 355.8,Z 295.998,A -85,B 0,C 180,E1 -13797.714,E2 -13797.714} C_VEL
LIN {X 0,Y 352.818,Z 283.444,A -85,B 0,C 180,E1 -13800.685,E2 -13800.685} C_VEL
LIN {X 0,Y 349.362,Z 270.275,A -85,B 0,C 180,E1 -13803.992,E2 -13803.992} C_VEL
LIN {X 0,Y 347.794,Z 264.835,A -85,B 0,C 180,E1 -13805.517,E2 -13805.517} C_VEL
LIN {X 0,Y 347.753,Z 264.79,A -85,B 0,C 180,E1 -13808.792,E2 -13808.792} C_VEL
LIN {X 0,Y 347.78,Z 264.785,A -85,B 0,C 180,E1 -13811.825,E2 -13811.825} C_VEL
LIN {X 0,Y 347.793,Z 264.776,A -85,B 0,C 180,E1 -13815.011,E2 -13815.011} C_VEL
LIN {X 0,Y 347.747,Z 264.777,A -85,B 0,C 180,E1 -13818.397,E2 -13818.397} C_VEL
LIN {X 0,Y 347.77,Z 264.787,A -85,B 0,C 180,E1 -13822.011,E2 -13822.011} C_VEL
LIN {X 0,Y 347.74,Z 264.785,A -85,B 0,C 180,E1 -13825.536,E2 -13825.536} C_VEL
LIN {X 0,Y 347.76,Z 264.766,A -85,B 0,C 180,E1 -13829.653,E2 -13829.653} C_VEL
LIN {X 0,Y 347.848,Z 264.779,A -85,B 0,C 180,E1 -13832.744,E2 -13832.744} C_VEL
LIN {X 0,Y 347.783,Z 264.784,A -85,B 0,C 180,E1 -13836.162,E2 -13836.162} C_VEL
LIN {X 0,Y 347.812,Z 264.779,A -85,B 0,C 180,E1 -13839.91,E2 -13839.91} C_VEL
LIN {X 0,Y 347.861,Z 264.775,A -85,B 0,C 180,E1 -13842.359,E2 -13842.359} C_VEL
LIN {X 0,Y 347.892,Z 264.775,A -85,B 0,C 180,E1 -13845.971,E2 -13845.971} C_VEL
LIN {X 0,Y 347.923,Z 264.767,A -85,B 0,C 180,E1 -13849.526,E2 -13849.526} C_VEL
LIN {X 0,Y 348.087,Z 264.739,A -85,B 0,C 180,E1 -13853.042,E2 -13853.042} C_VEL
LIN {X 0,Y 348.203,Z 264.728,A -85,B 0,C 180,E1 -13857.687,E2 -13857.687} C_VEL
LIN {X 0,Y 348.341,Z 264.719,A -85,B 0,C 180,E1 -13860,E2 -13860} C_VEL
LIN {X 0,Y 348.203,Z 264.725,A -85,B 0,C 180,E1 -13862.314,E2 -13862.314} C_VEL
LIN {X 0,Y 348.101,Z 264.739,A -85,B 0,C 180,E1 -13866.958,E2 -13866.958} C_VEL
LIN {X 0,Y 347.963,Z 264.768,A -85,B 0,C 180,E1 -13869.299,E2 -13869.299} C_VEL
LIN {X 0,Y 347.885,Z 264.771,A -85,B 0,C 180,E1 -13872.84,E2 -13872.84} C_VEL
LIN {X 0,Y 347.835,Z 264.774,A -85,B 0,C 180,E1 -13876.432,E2 -13876.432} C_VEL
LIN {X 0,Y 347.847,Z 264.78,A -85,B 0,C 180,E1 -13878.861,E2 -13878.861} C_VEL
LIN {X 0,Y 347.772,Z 264.79,A -85,B 0,C 180,E1 -13882.58,E2 -13882.58} C_VEL
LIN {X 0,Y 347.809,Z 264.785,A -85,B 0,C 180,E1 -13885.109,E2 -13885.109} C_VEL
LIN {X 0,Y 347.805,Z 264.772,A -85,B 0,C 180,E1 -13887.695,E2 -13887.695} C_VEL
LIN {X 0,Y 347.746,Z 264.779,A -85,B 0,C 180,E1 -13890.349,E2 -13890.349} C_VEL
LIN {X 0,Y 347.746,Z 264.78,A -85,B 0,C 180,E1 -13894.045,E2 -13894.045} C_VEL
LIN {X 0,Y 347.764,Z 264.793,A -85,B 0,C 180,E1 -13897.321,E2 -13897.321} C_VEL
LIN {X 0,Y 347.731,Z 264.778,A -85,B 0,C 180,E1 -13900.298,E2 -13900.298} C_VEL
LIN {X 0,Y 347.723,Z 264.787,A -85,B 0,C 180,E1 -13903.409,E2 -13903.409} C_VEL
LIN {X 0,Y 347.726,Z 264.792,A -85,B 0,C 180,E1 -13906.687,E2 -13906.687} C_VEL
LIN {X 0,Y 347.748,Z 264.774,A -85,B 0,C 180,E1 -13910.174,E2 -13910.174} C_VEL
LIN {X 0,Y 347.802,Z 264.964,A -85,B 0,C 180,E1 -13912.224,E2 -13912.224} C_VEL
LIN {X 0,Y 350.975,Z 276.729,A -85,B 0,C 180,E1 -13915.535,E2 -13915.535} C_VEL
LIN {X 0,Y 353.96,Z 289.711,A -85,B 0,C 180,E1 -13918.92,E2 -13918.92} C_VEL
LIN {X 0,Y 355.241,Z 296.141,A -85,B 0,C 180,E1 -13920.516,E2 -13920.516} C_VEL
LIN {X 0,Y 353.759,Z 308.668,A -85,B 0,C 180,E1 -13923.222,E2 -13923.222} C_VEL
LIN {X 0,Y 353.467,Z 311.814,A -85,B 0,C 180,E1 -13923.823,E2 -13923.823} C_VEL
LIN {X 0,Y 359.757,Z 345.113,A -85,B 0,C 180,E1 -13925.022,E2 -13925.022} C_VEL
LIN {X 0,Y 360.04,Z 349.433,A -85,B 0,C 180,E1 -13925.131,E2 -13925.131} C_VEL
LIN {X 0,Y 358.498,Z 426.758,A -85,B 0,C 180,E1 -13926.611,E2 -13926.611} C_VEL
LIN {X 0,Y 357.726,Z 440.279,A -85,B 0,C 180,E1 -13927.091,E2 -13927.091} C_VEL
LIN {X 0,Y 356.917,Z 452.946,A -85,B 0,C 180,E1 -13927.783,E2 -13927.783} C_VEL
LIN {X 0,Y 355.707,Z 465.526,A -85,B 0,C 180,E1 -13928.713,E2 -13928.713} C_VEL
LIN {X 0,Y 354.314,Z 477.142,A -85,B 0,C 180,E1 -13929.84,E2 -13929.84} C_VEL
LIN {X 0,Y 352.777,Z 487.604,A -85,B 0,C 180,E1 -13931.112,E2 -13931.112} C_VEL
LIN {X 0,Y 351.422,Z 497.063,A -85,B 0,C 180,E1 -13932.544,E2 -13932.544} C_VEL
LIN {X 0,Y 350.183,Z 504.848,A -85,B 0,C 180,E1 -13933.982,E2 -13933.982} C_VEL
LIN {X 0,Y 349.068,Z 512.525,A -85,B 0,C 180,E1 -13935.722,E2 -13935.722} C_VEL
LIN {X 0,Y 348.288,Z 517.751,A -85,B 0,C 180,E1 -13937.176,E2 -13937.176} C_VEL
LIN {X 0,Y 347.433,Z 522.896,A -85,B 0,C 180,E1 -13938.921,E2 -13938.921} C_VEL
LIN {X 0,Y 346.92,Z 526.934,A -85,B 0,C 180,E1 -13940.673,E2 -13940.673} C_VEL
LIN {X 0,Y 346.683,Z 529.091,A -85,B 0,C 180,E1 -13941.842,E2 -13941.842} C_VEL
LIN {X 0,Y 346.352,Z 531.842,A -85,B 0,C 180,E1 -13943.876,E2 -13943.876} C_VEL
LIN {X 0,Y 346.258,Z 533.065,A -85,B 0,C 180,E1 -13945.343,E2 -13945.343} C_VEL
LIN {X 0,Y 346.129,Z 533.871,A -85,B 0,C 180,E1 -13947.673,E2 -13947.673} C_VEL
LIN {X 0,Y 346.148,Z 533.72,A -85,B 0,C 180,E1 -13948.837,E2 -13948.837} C_VEL
LIN {X 0,Y 346.228,Z 532.294,A -85,B 0,C 180,E1 -13951.163,E2 -13951.163} C_VEL
LIN {X 0,Y 346.507,Z 529.4,A -85,B 0,C 180,E1 -13953.488,E2 -13953.488} C_VEL
LIN {X 0,Y 346.832,Z 526.141,A -85,B 0,C 180,E1 -13955.232,E2 -13955.232} C_VEL
LIN {X 0,Y 347.375,Z 521.881,A -85,B 0,C 180,E1 -13956.972,E2 -13956.972} C_VEL
LIN {X 0,Y 348.143,Z 515.52,A -85,B 0,C 180,E1 -13959.001,E2 -13959.001} C_VEL
LIN {X 0,Y 349.046,Z 508.601,A -85,B 0,C 180,E1 -13960.734,E2 -13960.734} C_VEL
LIN {X 0,Y 350.3,Z 500.022,A -85,B 0,C 180,E1 -13962.455,E2 -13962.455} C_VEL
LIN {X 0,Y 351.445,Z 491.289,A -85,B 0,C 180,E1 -13963.884,E2 -13963.884} C_VEL
LIN {X 0,Y 352.638,Z 481.74,A -85,B 0,C 180,E1 -13965.163,E2 -13965.163} C_VEL
LIN {X 0,Y 353.802,Z 471.339,A -85,B 0,C 180,E1 -13966.295,E2 -13966.295} C_VEL
LIN {X 0,Y 354.997,Z 459.936,A -85,B 0,C 180,E1 -13967.275,E2 -13967.275} C_VEL
LIN {X 0,Y 355.988,Z 448.241,A -85,B 0,C 180,E1 -13968.041,E2 -13968.041} C_VEL
LIN {X 0,Y 356.69,Z 435.492,A -85,B 0,C 180,E1 -13968.646,E2 -13968.646} C_VEL
LIN {X 0,Y 357.244,Z 421.586,A -85,B 0,C 180,E1 -13969.052,E2 -13969.052} C_VEL
LIN {X 0,Y 357.93,Z 382.612,A -85,B 0,C 180,E1 -13969.787,E2 -13969.787} C_VEL
LIN {X 0,Y 357.257,Z 376.815,A -85,B 0,C 180,E1 -13969.946,E2 -13969.946} C_VEL
LIN {X 0,Y 352.399,Z 358.111,A -85,B 0,C 180,E1 -13970.652,E2 -13970.652} C_VEL
LIN {X 0,Y 351.921,Z 352.307,A -85,B 0,C 180,E1 -13970.804,E2 -13970.804} C_VEL
LIN {X 0,Y 351.794,Z 346.18,A -85,B 0,C 180,E1 -13970.939,E2 -13970.939} C_VEL
LIN {X 0,Y 346.69,Z 316.307,A -85,B 0,C 180,E1 -13971.931,E2 -13971.931} C_VEL
LIN {X 0,Y 345.846,Z 311.392,A -85,B 0,C 180,E1 -13972.145,E2 -13972.145} C_VEL
LIN {X 0,Y 347.65,Z 296.059,A -85,B 0,C 180,E1 -13975.441,E2 -13975.441} C_VEL
LIN {X 0,Y 345.542,Z 284.963,A -85,B 0,C 180,E1 -13978.218,E2 -13978.218} C_VEL
LIN {X 0,Y 342.817,Z 273.821,A -85,B 0,C 180,E1 -13981.174,E2 -13981.174} C_VEL
LIN {X 0,Y 340.723,Z 265.734,A -85,B 0,C 180,E1 -13983.487,E2 -13983.487} C_VEL
LIN {X 0,Y 340.706,Z 265.669,A -85,B 0,C 180,E1 -13986.741,E2 -13986.741} C_VEL
LIN {X 0,Y 340.688,Z 265.666,A -85,B 0,C 180,E1 -13990.246,E2 -13990.246} C_VEL
LIN {X 0,Y 340.652,Z 265.673,A -85,B 0,C 180,E1 -13993.772,E2 -13993.772} C_VEL
LIN {X 0,Y 340.697,Z 265.67,A -85,B 0,C 180,E1 -13997.954,E2 -13997.954} C_VEL
LIN {X 0,Y 340.731,Z 265.661,A -85,B 0,C 180,E1 -14001.772,E2 -14001.772} C_VEL
LIN {X 0,Y 340.72,Z 265.644,A -85,B 0,C 180,E1 -14005.594,E2 -14005.594} C_VEL
LIN {X 0,Y 340.701,Z 265.668,A -85,B 0,C 180,E1 -14008.955,E2 -14008.955} C_VEL
LIN {X 0,Y 340.776,Z 265.655,A -85,B 0,C 180,E1 -14012.473,E2 -14012.473} C_VEL
LIN {X 0,Y 340.751,Z 265.654,A -85,B 0,C 180,E1 -14015.637,E2 -14015.637} C_VEL
LIN {X 0,Y 340.74,Z 265.659,A -85,B 0,C 180,E1 -14019.473,E2 -14019.473} C_VEL
LIN {X 0,Y 340.853,Z 265.649,A -85,B 0,C 180,E1 -14021.983,E2 -14021.983} C_VEL
LIN {X 0,Y 340.865,Z 265.642,A -85,B 0,C 180,E1 -14025.704,E2 -14025.704} C_VEL
LIN {X 0,Y 340.865,Z 265.641,A -85,B 0,C 180,E1 -14029.306,E2 -14029.306} C_VEL
LIN {X 0,Y 341.054,Z 265.627,A -85,B 0,C 180,E1 -14032.897,E2 -14032.897} C_VEL
LIN {X 0,Y 341.164,Z 265.611,A -85,B 0,C 180,E1 -14037.638,E2 -14037.638} C_VEL
LIN {X 0,Y 341.29,Z 265.59,A -85,B 0,C 180,E1 -14040,E2 -14040} C_VEL
LIN {X 0,Y 341.164,Z 265.61,A -85,B 0,C 180,E1 -14042.361,E2 -14042.361} C_VEL
LIN {X 0,Y 341.069,Z 265.62,A -85,B 0,C 180,E1 -14047.102,E2 -14047.102} C_VEL
LIN {X 0,Y 340.864,Z 265.639,A -85,B 0,C 180,E1 -14050.694,E2 -14050.694} C_VEL
LIN {X 0,Y 340.857,Z 265.65,A -85,B 0,C 180,E1 -14054.325,E2 -14054.325} C_VEL
LIN {X 0,Y 340.831,Z 265.655,A -85,B 0,C 180,E1 -14058.466,E2 -14058.466} C_VEL
LIN {X 0,Y 340.748,Z 265.662,A -85,B 0,C 180,E1 -14061.857,E2 -14061.857} C_VEL
LIN {X 0,Y 340.767,Z 265.657,A -85,B 0,C 180,E1 -14065.664,E2 -14065.664} C_VEL
LIN {X 0,Y 340.737,Z 265.657,A -85,B 0,C 180,E1 -14068.32,E2 -14068.32} C_VEL
LIN {X 0,Y 340.699,Z 265.646,A -85,B 0,C 180,E1 -14071.044,E2 -14071.044} C_VEL
LIN {X 0,Y 340.713,Z 265.662,A -85,B 0,C 180,E1 -14075.279,E2 -14075.279} C_VEL
LIN {X 0,Y 340.706,Z 265.663,A -85,B 0,C 180,E1 -14078.387,E2 -14078.387} C_VEL
LIN {X 0,Y 340.694,Z 265.656,A -85,B 0,C 180,E1 -14082.046,E2 -14082.046} C_VEL
LIN {X 0,Y 340.68,Z 265.663,A -85,B 0,C 180,E1 -14085.462,E2 -14085.462} C_VEL
LIN {X 0,Y 340.681,Z 265.624,A -85,B 0,C 180,E1 -14088.691,E2 -14088.691} C_VEL
LIN {X 0,Y 340.73,Z 265.667,A -85,B 0,C 180,E1 -14091.773,E2 -14091.773} C_VEL
LIN {X 0,Y 340.784,Z 265.866,A -85,B 0,C 180,E1 -14094.998,E2 -14094.998} C_VEL
LIN {X 0,Y 344.13,Z 278.353,A -85,B 0,C 180,E1 -14098.219,E2 -14098.219} C_VEL
LIN {X 0,Y 347.166,Z 290.984,A -85,B 0,C 180,E1 -14101.263,E2 -14101.263} C_VEL
LIN {X 0,Y 348.576,Z 297.831,A -85,B 0,C 180,E1 -14102.837,E2 -14102.837} C_VEL
LIN {X 0,Y 348.539,Z 299.721,A -85,B 0,C 180,E1 -14103.128,E2 -14103.128} C_VEL
LIN {X 0,Y 352.905,Z 328.398,A -85,B 0,C 180,E1 -14104.12,E2 -14104.12} C_VEL
LIN {X 0,Y 350.436,Z 430.86,A -85,B 0,C 180,E1 -14106.314,E2 -14106.314} C_VEL
LIN {X 0,Y 349.606,Z 445.362,A -85,B 0,C 180,E1 -14106.843,E2 -14106.843} C_VEL
LIN {X 0,Y 348.54,Z 459.798,A -85,B 0,C 180,E1 -14107.63,E2 -14107.63} C_VEL
LIN {X 0,Y 347.336,Z 473.466,A -85,B 0,C 180,E1 -14108.641,E2 -14108.641} C_VEL
LIN {X 0,Y 346.021,Z 485.719,A -85,B 0,C 180,E1 -14109.801,E2 -14109.801} C_VEL
LIN {X 0,Y 344.417,Z 497.986,A -85,B 0,C 180,E1 -14111.254,E2 -14111.254} C_VEL
LIN {X 0,Y 343.148,Z 508.087,A -85,B 0,C 180,E1 -14112.724,E2 -14112.724} C_VEL
LIN {X 0,Y 341.958,Z 518.113,A -85,B 0,C 180,E1 -14114.504,E2 -14114.504} C_VEL
LIN {X 0,Y 341.075,Z 526.392,A -85,B 0,C 180,E1 -14116.293,E2 -14116.293} C_VEL
LIN {X 0,Y 340.144,Z 534.274,A -85,B 0,C 180,E1 -14118.378,E2 -14118.378} C_VEL
LIN {X 0,Y 339.568,Z 540.554,A -85,B 0,C 180,E1 -14120.47,E2 -14120.47} C_VEL
LIN {X 0,Y 339.283,Z 544.789,A -85,B 0,C 180,E1 -14122.262,E2 -14122.262} C_VEL
LIN {X 0,Y 339.083,Z 548.326,A -85,B 0,C 180,E1 -14124.193,E2 -14124.193} C_VEL
LIN {X 0,Y 339.055,Z 551.172,A -85,B 0,C 180,E1 -14126.435,E2 -14126.435} C_VEL
LIN {X 0,Y 339.016,Z 552.777,A -85,B 0,C 180,E1 -14128.812,E2 -14128.812} C_VEL
LIN {X 0,Y 339.065,Z 553.046,A -85,B 0,C 180,E1 -14130,E2 -14130} C_VEL
LIN {X 0,Y 338.994,Z 552.511,A -85,B 0,C 180,E1 -14132.376,E2 -14132.376} C_VEL
LIN {X 0,Y 339.056,Z 551.71,A -85,B 0,C 180,E1 -14133.565,E2 -14133.565} C_VEL
LIN {X 0,Y 339.132,Z 548.988,A -85,B 0,C 180,E1 -14135.947,E2 -14135.947} C_VEL
LIN {X 0,Y 339.375,Z 544.738,A -85,B 0,C 180,E1 -14138.335,E2 -14138.335} C_VEL
LIN {X 0,Y 339.751,Z 540.509,A -85,B 0,C 180,E1 -14140.127,E2 -14140.127} C_VEL
LIN {X 0,Y 340.525,Z 534.253,A -85,B 0,C 180,E1 -14142.213,E2 -14142.213} C_VEL
LIN {X 0,Y 341.537,Z 526.406,A -85,B 0,C 180,E1 -14144.296,E2 -14144.296} C_VEL
LIN {X 0,Y 342.556,Z 518.179,A -85,B 0,C 180,E1 -14146.079,E2 -14146.079} C_VEL
LIN {X 0,Y 343.957,Z 508.227,A -85,B 0,C 180,E1 -14147.848,E2 -14147.848} C_VEL
LIN {X 0,Y 345.548,Z 497.133,A -85,B 0,C 180,E1 -14149.453,E2 -14149.453} C_VEL
LIN {X 0,Y 347.036,Z 486.072,A -85,B 0,C 180,E1 -14150.756,E2 -14150.756} C_VEL
LIN {X 0,Y 348.497,Z 473.263,A -85,B 0,C 180,E1 -14151.971,E2 -14151.971} C_VEL
LIN {X 0,Y 349.746,Z 460.566,A -85,B 0,C 180,E1 -14152.913,E2 -14152.913} C_VEL
LIN {X 0,Y 350.961,Z 446.493,A -85,B 0,C 180,E1 -14153.687,E2 -14153.687} C_VEL
LIN {X 0,Y 351.823,Z 432.657,A -85,B 0,C 180,E1 -14154.213,E2 -14154.213} C_VEL
LIN {X 0,Y 352.85,Z 397.773,A -85,B 0,C 180,E1 -14154.989,E2 -14154.989} C_VEL
LIN {X 0,Y 354.44,Z 328.25,A -85,B 0,C 180,E1 -14156.478,E2 -14156.478} C_VEL
LIN {X 0,Y 349.904,Z 301.301,A -85,B 0,C 180,E1 -14157.477,E2 -14157.477} C_VEL
LIN {X 0,Y 349.262,Z 299.077,A -85,B 0,C 180,E1 -14157.649,E2 -14157.649} C_VEL
LIN {X 0,Y 346.552,Z 287.281,A -85,B 0,C 180,E1 -14160.463,E2 -14160.463} C_VEL
LIN {X 0,Y 343.132,Z 273.985,A -85,B 0,C 180,E1 -14163.853,E2 -14163.853} C_VEL
LIN {X 0,Y 340.736,Z 265.725,A -85,B 0,C 180,E1 -14166.165,E2 -14166.165} C_VEL
LIN {X 0,Y 340.731,Z 265.664,A -85,B 0,C 180,E1 -14169.747,E2 -14169.747} C_VEL
LIN {X 0,Y 340.737,Z 265.667,A -85,B 0,C 180,E1 -14172.894,E2 -14172.894} C_VEL
LIN {X 0,Y 340.673,Z 265.675,A -85,B 0,C 180,E1 -14176.222,E2 -14176.222} C_VEL
LIN {X 0,Y 340.684,Z 265.661,A -85,B 0,C 180,E1 -14179.753,E2 -14179.753} C_VEL
LIN {X 0,Y 340.701,Z 265.652,A -85,B 0,C 180,E1 -14183.258,E2 -14183.258} C_VEL
LIN {X 0,Y 340.688,Z 265.669,A -85,B 0,C 180,E1 -14186.153,E2 -14186.153} C_VEL
LIN {X 0,Y 340.77,Z 265.634,A -85,B 0,C 180,E1 -14190.332,E2 -14190.332} C_VEL
LIN {X 0,Y 340.8,Z 265.656,A -85,B 0,C 180,E1 -14193.02,E2 -14193.02} C_VEL
LIN {X 0,Y 340.724,Z 265.666,A -85,B 0,C 180,E1 -14196.927,E2 -14196.927} C_VEL
LIN {X 0,Y 340.789,Z 265.657,A -85,B 0,C 180,E1 -14200.734,E2 -14200.734} C_VEL
LIN {X 0,Y 340.781,Z 265.654,A -85,B 0,C 180,E1 -14203.219,E2 -14203.219} C_VEL
LIN {X 0,Y 340.838,Z 265.65,A -85,B 0,C 180,E1 -14206.891,E2 -14206.891} C_VEL
LIN {X 0,Y 340.921,Z 265.642,A -85,B 0,C 180,E1 -14210.508,E2 -14210.508} C_VEL
LIN {X 0,Y 341.055,Z 265.614,A -85,B 0,C 180,E1 -14212.898,E2 -14212.898} C_VEL
LIN {X 0,Y 341.164,Z 265.604,A -85,B 0,C 180,E1 -14217.639,E2 -14217.639} C_VEL
LIN {X 0,Y 341.291,Z 265.597,A -85,B 0,C 180,E1 -14220,E2 -14220} C_VEL
LIN {X 0,Y 341.165,Z 265.601,A -85,B 0,C 180,E1 -14222.362,E2 -14222.362} C_VEL
LIN {X 0,Y 341.07,Z 265.615,A -85,B 0,C 180,E1 -14227.102,E2 -14227.102} C_VEL
LIN {X 0,Y 340.866,Z 265.646,A -85,B 0,C 180,E1 -14230.694,E2 -14230.694} C_VEL
LIN {X 0,Y 340.859,Z 265.649,A -85,B 0,C 180,E1 -14234.325,E2 -14234.325} C_VEL
LIN {X 0,Y 340.833,Z 265.653,A -85,B 0,C 180,E1 -14238.467,E2 -14238.467} C_VEL
LIN {X 0,Y 340.75,Z 265.664,A -85,B 0,C 180,E1 -14241.858,E2 -14241.858} C_VEL
LIN {X 0,Y 340.77,Z 265.663,A -85,B 0,C 180,E1 -14245.665,E2 -14245.665} C_VEL
LIN {X 0,Y 340.725,Z 265.645,A -85,B 0,C 180,E1 -14248.322,E2 -14248.322} C_VEL
LIN {X 0,Y 340.695,Z 265.665,A -85,B 0,C 180,E1 -14251.046,E2 -14251.046} C_VEL
LIN {X 0,Y 340.717,Z 265.649,A -85,B 0,C 180,E1 -14255.28,E2 -14255.28} C_VEL
LIN {X 0,Y 340.711,Z 265.667,A -85,B 0,C 180,E1 -14258.387,E2 -14258.387} C_VEL
LIN {X 0,Y 340.698,Z 265.672,A -85,B 0,C 180,E1 -14262.046,E2 -14262.046} C_VEL
LIN {X 0,Y 340.653,Z 265.679,A -85,B 0,C 180,E1 -14266.228,E2 -14266.228} C_VEL
LIN {X 0,Y 340.69,Z 265.662,A -85,B 0,C 180,E1 -14269.754,E2 -14269.754} C_VEL
LIN {X 0,Y 340.749,Z 265.81,A -85,B 0,C 180,E1 -14271.561,E2 -14271.561} C_VEL
LIN {X 0,Y 344.088,Z 278.087,A -85,B 0,C 180,E1 -14275.118,E2 -14275.118} C_VEL
LIN {X 0,Y 347.082,Z 291.063,A -85,B 0,C 180,E1 -14278.583,E2 -14278.583} C_VEL
LIN {X 0,Y 348.463,Z 298.274,A -85,B 0,C 180,E1 -14280.407,E2 -14280.407} C_VEL
LIN {X 0,Y 346.822,Z 311.439,A -85,B 0,C 180,E1 -14283.253,E2 -14283.253} C_VEL
LIN {X 0,Y 352.471,Z 341.172,A -85,B 0,C 180,E1 -14284.381,E2 -14284.381} C_VEL
LIN {X 0,Y 353.631,Z 348.827,A -85,B 0,C 180,E1 -14284.631,E2 -14284.631} C_VEL
LIN {X 0,Y 352.005,Z 426.889,A -85,B 0,C 180,E1 -14286.153,E2 -14286.153} C_VEL
LIN {X 0,Y 351.212,Z 440.44,A -85,B 0,C 180,E1 -14286.643,E2 -14286.643} C_VEL
LIN {X 0,Y 350.307,Z 453.673,A -85,B 0,C 180,E1 -14287.383,E2 -14287.383} C_VEL
LIN {X 0,Y 349.109,Z 465.624,A -85,B 0,C 180,E1 -14288.29,E2 -14288.29} C_VEL
LIN {X 0,Y 347.652,Z 477.243,A -85,B 0,C 180,E1 -14289.437,E2 -14289.437} C_VEL
LIN {X 0,Y 346.077,Z 487.711,A -85,B 0,C 180,E1 -14290.732,E2 -14290.732} C_VEL
LIN {X 0,Y 344.626,Z 497.178,A -85,B 0,C 180,E1 -14292.188,E2 -14292.188} C_VEL
LIN {X 0,Y 343.34,Z 504.968,A -85,B 0,C 180,E1 -14293.653,E2 -14293.653} C_VEL
LIN {X 0,Y 342.174,Z 512.227,A -85,B 0,C 180,E1 -14295.316,E2 -14295.316} C_VEL
LIN {X 0,Y 341.331,Z 517.89,A -85,B 0,C 180,E1 -14296.91,E2 -14296.91} C_VEL
LIN {X 0,Y 340.431,Z 523.045,A -85,B 0,C 180,E1 -14298.69,E2 -14298.69} C_VEL
LIN {X 0,Y 339.893,Z 527.091,A -85,B 0,C 180,E1 -14300.479,E2 -14300.479} C_VEL
LIN {X 0,Y 339.639,Z 529.254,A -85,B 0,C 180,E1 -14301.672,E2 -14301.672} C_VEL
LIN {X 0,Y 339.256,Z 532.181,A -85,B 0,C 180,E1 -14303.921,E2 -14303.921} C_VEL
LIN {X 0,Y 339.175,Z 533.249,A -85,B 0,C 180,E1 -14305.246,E2 -14305.246} C_VEL
LIN {X 0,Y 339.041,Z 534.067,A -85,B 0,C 180,E1 -14307.624,E2 -14307.624} C_VEL
LIN {X 0,Y 339.05,Z 533.927,A -85,B 0,C 180,E1 -14308.812,E2 -14308.812} C_VEL
LIN {X 0,Y 339.134,Z 532.516,A -85,B 0,C 180,E1 -14311.187,E2 -14311.187} C_VEL
LIN {X 0,Y 339.43,Z 529.636,A -85,B 0,C 180,E1 -14313.561,E2 -14313.561} C_VEL
LIN {X 0,Y 339.786,Z 526.393,A -85,B 0,C 180,E1 -14315.34,E2 -14315.34} C_VEL
LIN {X 0,Y 340.443,Z 521.412,A -85,B 0,C 180,E1 -14317.396,E2 -14317.396} C_VEL
LIN {X 0,Y 341.261,Z 514.748,A -85,B 0,C 180,E1 -14319.483,E2 -14319.483} C_VEL
LIN {X 0,Y 342.298,Z 507.61,A -85,B 0,C 180,E1 -14321.248,E2 -14321.248} C_VEL
LIN {X 0,Y 343.623,Z 498.795,A -85,B 0,C 180,E1 -14323.001,E2 -14323.001} C_VEL
LIN {X 0,Y 344.858,Z 489.782,A -85,B 0,C 180,E1 -14324.456,E2 -14324.456} C_VEL
LIN {X 0,Y 346.117,Z 479.866,A -85,B 0,C 180,E1 -14325.758,E2 -14325.758} C_VEL
LIN {X 0,Y 347.339,Z 468.926,A -85,B 0,C 180,E1 -14326.909,E2 -14326.909} C_VEL
LIN {X 0,Y 348.43,Z 458.708,A -85,B 0,C 180,E1 -14327.762,E2 -14327.762} C_VEL
LIN {X 0,Y 349.482,Z 446.548,A -85,B 0,C 180,E1 -14328.541,E2 -14328.541} C_VEL
LIN {X 0,Y 350.213,Z 433.318,A -85,B 0,C 180,E1 -14329.145,E2 -14329.145} C_VEL
LIN {X 0,Y 350.679,Z 420.994,A -85,B 0,C 180,E1 -14329.489,E2 -14329.489} C_VEL
LIN {X 0,Y 351.921,Z 352.307,A -85,B 0,C 180,E1 -14330.804,E2 -14330.804} C_VEL
LIN {X 0,Y 351.572,Z 348.465,A -85,B 0,C 180,E1 -14330.907,E2 -14330.907} C_VEL
LIN {X 0,Y 349.883,Z 342.988,A -85,B 0,C 180,E1 -14331.14,E2 -14331.14} C_VEL
LIN {X 0,Y 343.091,Z 329.196,A -85,B 0,C 180,E1 -14331.93,E2 -14331.93} C_VEL
LIN {X 0,Y 341.386,Z 323.61,A -85,B 0,C 180,E1 -14332.179,E2 -14332.179} C_VEL
LIN {X 0,Y 339.167,Z 311.45,A -85,B 0,C 180,E1 -14332.645,E2 -14332.645} C_VEL
LIN {X 0,Y 340.832,Z 297.582,A -85,B 0,C 180,E1 -14335.659,E2 -14335.659} C_VEL
LIN {X 0,Y 338.685,Z 286.462,A -85,B 0,C 180,E1 -14338.507,E2 -14338.507} C_VEL
LIN {X 0,Y 335.633,Z 274.055,A -85,B 0,C 180,E1 -14341.887,E2 -14341.887} C_VEL
LIN {X 0,Y 333.699,Z 266.635,A -85,B 0,C 180,E1 -14344.061,E2 -14344.061} C_VEL
LIN {X 0,Y 333.653,Z 266.541,A -85,B 0,C 180,E1 -14347.65,E2 -14347.65} C_VEL
LIN {X 0,Y 333.647,Z 266.539,A -85,B 0,C 180,E1 -14350.766,E2 -14350.766} C_VEL
LIN {X 0,Y 333.593,Z 266.546,A -85,B 0,C 180,E1 -14354.249,E2 -14354.249} C_VEL
LIN {X 0,Y 333.64,Z 266.551,A -85,B 0,C 180,E1 -14357.617,E2 -14357.617} C_VEL
LIN {X 0,Y 333.651,Z 266.533,A -85,B 0,C 180,E1 -14361.201,E2 -14361.201} C_VEL
LIN {X 0,Y 333.674,Z 266.543,A -85,B 0,C 180,E1 -14363.86,E2 -14363.86} C_VEL
LIN {X 0,Y 333.641,Z 266.529,A -85,B 0,C 180,E1 -14367.412,E2 -14367.412} C_VEL
LIN {X 0,Y 333.708,Z 266.536,A -85,B 0,C 180,E1 -14371.027,E2 -14371.027} C_VEL
LIN {X 0,Y 333.732,Z 266.538,A -85,B 0,C 180,E1 -14373.753,E2 -14373.753} C_VEL
LIN {X 0,Y 333.716,Z 266.54,A -85,B 0,C 180,E1 -14377.913,E2 -14377.913} C_VEL
LIN {X 0,Y 333.789,Z 266.529,A -85,B 0,C 180,E1 -14381.589,E2 -14381.589} C_VEL
LIN {X 0,Y 333.804,Z 266.521,A -85,B 0,C 180,E1 -14385.576,E2 -14385.576} C_VEL
LIN {X 0,Y 333.828,Z 266.519,A -85,B 0,C 180,E1 -14389.077,E2 -14389.077} C_VEL
LIN {X 0,Y 334.001,Z 266.507,A -85,B 0,C 180,E1 -14392.747,E2 -14392.747} C_VEL
LIN {X 0,Y 333.804,Z 266.516,A -85,B 0,C 180,E1 -14395.169,E2 -14395.169} C_VEL
LIN {X 0,Y 334.101,Z 266.491,A -85,B 0,C 180,E1 -14397.588,E2 -14397.588} C_VEL
LIN {X 0,Y 334.241,Z 266.467,A -85,B 0,C 180,E1 -14400,E2 -14400} C_VEL
LIN {X 0,Y 334.101,Z 266.49,A -85,B 0,C 180,E1 -14402.411,E2 -14402.411} C_VEL
LIN {X 0,Y 334.019,Z 266.498,A -85,B 0,C 180,E1 -14407.252,E2 -14407.252} C_VEL
LIN {X 0,Y 333.827,Z 266.515,A -85,B 0,C 180,E1 -14410.922,E2 -14410.922} C_VEL
LIN {X 0,Y 333.802,Z 266.525,A -85,B 0,C 180,E1 -14414.634,E2 -14414.634} C_VEL
LIN {X 0,Y 333.79,Z 266.53,A -85,B 0,C 180,E1 -14418.655,E2 -14418.655} C_VEL
LIN {X 0,Y 333.687,Z 266.546,A -85,B 0,C 180,E1 -14422.278,E2 -14422.278} C_VEL
LIN {X 0,Y 333.731,Z 266.54,A -85,B 0,C 180,E1 -14426.246,E2 -14426.246} C_VEL
LIN {X 0,Y 333.706,Z 266.526,A -85,B 0,C 180,E1 -14428.972,E2 -14428.972} C_VEL
LIN {X 0,Y 333.641,Z 266.545,A -85,B 0,C 180,E1 -14432.588,E2 -14432.588} C_VEL
LIN {X 0,Y 333.671,Z 266.526,A -85,B 0,C 180,E1 -14436.139,E2 -14436.139} C_VEL
LIN {X 0,Y 333.643,Z 266.551,A -85,B 0,C 180,E1 -14439.193,E2 -14439.193} C_VEL
LIN {X 0,Y 333.628,Z 266.537,A -85,B 0,C 180,E1 -14442.5,E2 -14442.5} C_VEL
LIN {X 0,Y 333.618,Z 266.532,A -85,B 0,C 180,E1 -14445.96,E2 -14445.96} C_VEL
LIN {X 0,Y 333.643,Z 266.506,A -85,B 0,C 180,E1 -14449.316,E2 -14449.316} C_VEL
LIN {X 0,Y 333.662,Z 266.519,A -85,B 0,C 180,E1 -14453.168,E2 -14453.168} C_VEL
LIN {X 0,Y 333.723,Z 266.809,A -85,B 0,C 180,E1 -14454.399,E2 -14454.399} C_VEL
LIN {X 0,Y 337.294,Z 280.036,A -85,B 0,C 180,E1 -14457.906,E2 -14457.906} C_VEL
LIN {X 0,Y 340.296,Z 292.527,A -85,B 0,C 180,E1 -14460.995,E2 -14460.995} C_VEL
LIN {X 0,Y 341.779,Z 299.531,A -85,B 0,C 180,E1 -14462.591,E2 -14462.591} C_VEL
LIN {X 0,Y 343.935,Z 312.316,A -85,B 0,C 180,E1 -14463.088,E2 -14463.088} C_VEL
LIN {X 0,Y 346.385,Z 329.764,A -85,B 0,C 180,E1 -14463.678,E2 -14463.678} C_VEL
LIN {X 0,Y 343.822,Z 431.771,A -85,B 0,C 180,E1 -14465.91,E2 -14465.91} C_VEL
LIN {X 0,Y 342.951,Z 445.937,A -85,B 0,C 180,E1 -14466.447,E2 -14466.447} C_VEL
LIN {X 0,Y 341.853,Z 460.209,A -85,B 0,C 180,E1 -14467.248,E2 -14467.248} C_VEL
LIN {X 0,Y 340.579,Z 473.991,A -85,B 0,C 180,E1 -14468.296,E2 -14468.296} C_VEL
LIN {X 0,Y 339.159,Z 486.58,A -85,B 0,C 180,E1 -14469.533,E2 -14469.533} C_VEL
LIN {X 0,Y 337.499,Z 498.664,A -85,B 0,C 180,E1 -14471.012,E2 -14471.012} C_VEL
LIN {X 0,Y 336.074,Z 509.536,A -85,B 0,C 180,E1 -14472.663,E2 -14472.663} C_VEL
LIN {X 0,Y 334.895,Z 519.253,A -85,B 0,C 180,E1 -14474.471,E2 -14474.471} C_VEL
LIN {X 0,Y 333.948,Z 527.347,A -85,B 0,C 180,E1 -14476.305,E2 -14476.305} C_VEL
LIN {X 0,Y 333.018,Z 535.005,A -85,B 0,C 180,E1 -14478.435,E2 -14478.435} C_VEL
LIN {X 0,Y 332.502,Z 540.292,A -85,B 0,C 180,E1 -14480.265,E2 -14480.265} C_VEL
LIN {X 0,Y 332.202,Z 544.544,A -85,B 0,C 180,E1 -14482.096,E2 -14482.096} C_VEL
LIN {X 0,Y 331.987,Z 548.366,A -85,B 0,C 180,E1 -14484.247,E2 -14484.247} C_VEL
LIN {X 0,Y 331.957,Z 550.954,A -85,B 0,C 180,E1 -14486.359,E2 -14486.359} C_VEL
LIN {X 0,Y 331.922,Z 552.571,A -85,B 0,C 180,E1 -14488.787,E2 -14488.787} C_VEL
LIN {X 0,Y 331.968,Z 552.844,A -85,B 0,C 180,E1 -14490,E2 -14490} C_VEL
LIN {X 0,Y 331.911,Z 552.319,A -85,B 0,C 180,E1 -14492.427,E2 -14492.427} C_VEL
LIN {X 0,Y 331.959,Z 551.524,A -85,B 0,C 180,E1 -14493.642,E2 -14493.642} C_VEL
LIN {X 0,Y 332.041,Z 548.811,A -85,B 0,C 180,E1 -14496.075,E2 -14496.075} C_VEL
LIN {X 0,Y 332.311,Z 544.569,A -85,B 0,C 180,E1 -14498.513,E2 -14498.513} C_VEL
LIN {X 0,Y 332.716,Z 540.345,A -85,B 0,C 180,E1 -14500.343,E2 -14500.343} C_VEL
LIN {X 0,Y 333.542,Z 534.095,A -85,B 0,C 180,E1 -14502.473,E2 -14502.473} C_VEL
LIN {X 0,Y 334.614,Z 526.252,A -85,B 0,C 180,E1 -14504.598,E2 -14504.598} C_VEL
LIN {X 0,Y 335.678,Z 518.028,A -85,B 0,C 180,E1 -14506.418,E2 -14506.418} C_VEL
LIN {X 0,Y 337.164,Z 508.079,A -85,B 0,C 180,E1 -14508.22,E2 -14508.22} C_VEL
LIN {X 0,Y 338.82,Z 496.985,A -85,B 0,C 180,E1 -14509.856,E2 -14509.856} C_VEL
LIN {X 0,Y 340.389,Z 485.921,A -85,B 0,C 180,E1 -14511.181,E2 -14511.181} C_VEL
LIN {X 0,Y 341.857,Z 473.594,A -85,B 0,C 180,E1 -14512.376,E2 -14512.376} C_VEL
LIN {X 0,Y 343.213,Z 460.386,A -85,B 0,C 180,E1 -14513.374,E2 -14513.374} C_VEL
LIN {X 0,Y 344.483,Z 446.278,A -85,B 0,C 180,E1 -14514.161,E2 -14514.161} C_VEL
LIN {X 0,Y 345.353,Z 432.368,A -85,B 0,C 180,E1 -14514.696,E2 -14514.696} C_VEL
LIN {X 0,Y 346.653,Z 388.171,A -85,B 0,C 180,E1 -14515.685,E2 -14515.685} C_VEL
LIN {X 0,Y 347.998,Z 328.795,A -85,B 0,C 180,E1 -14516.983,E2 -14516.983} C_VEL
LIN {X 0,Y 343.72,Z 303.436,A -85,B 0,C 180,E1 -14517.951,E2 -14517.951} C_VEL
LIN {X 0,Y 342.208,Z 299.384,A -85,B 0,C 180,E1 -14518.229,E2 -14518.229} C_VEL
LIN {X 0,Y 339.148,Z 286.406,A -85,B 0,C 180,E1 -14521.422,E2 -14521.422} C_VEL
LIN {X 0,Y 335.829,Z 274.014,A -85,B 0,C 180,E1 -14524.718,E2 -14524.718} C_VEL
LIN {X 0,Y 333.668,Z 266.604,A -85,B 0,C 180,E1 -14526.869,E2 -14526.869} C_VEL
LIN {X 0,Y 333.696,Z 266.533,A -85,B 0,C 180,E1 -14530.759,E2 -14530.759} C_VEL
LIN {X 0,Y 333.666,Z 266.534,A -85,B 0,C 180,E1 -14534.264,E2 -14534.264} C_VEL
LIN {X 0,Y 333.639,Z 266.541,A -85,B 0,C 180,E1 -14537.618,E2 -14537.618} C_VEL
LIN {X 0,Y 333.649,Z 266.55,A -85,B 0,C 180,E1 -14541.202,E2 -14541.202} C_VEL
LIN {X 0,Y 333.672,Z 266.524,A -85,B 0,C 180,E1 -14543.861,E2 -14543.861} C_VEL
LIN {X 0,Y 333.639,Z 266.551,A -85,B 0,C 180,E1 -14547.413,E2 -14547.413} C_VEL
LIN {X 0,Y 333.707,Z 266.517,A -85,B 0,C 180,E1 -14551.028,E2 -14551.028} C_VEL
LIN {X 0,Y 333.731,Z 266.541,A -85,B 0,C 180,E1 -14553.754,E2 -14553.754} C_VEL
LIN {X 0,Y 333.715,Z 266.541,A -85,B 0,C 180,E1 -14557.914,E2 -14557.914} C_VEL
LIN {X 0,Y 333.789,Z 266.533,A -85,B 0,C 180,E1 -14561.59,E2 -14561.59} C_VEL
LIN {X 0,Y 333.803,Z 266.529,A -85,B 0,C 180,E1 -14565.577,E2 -14565.577} C_VEL
LIN {X 0,Y 333.828,Z 266.519,A -85,B 0,C 180,E1 -14569.078,E2 -14569.078} C_VEL
LIN {X 0,Y 334.008,Z 266.492,A -85,B 0,C 180,E1 -14572.748,E2 -14572.748} C_VEL
LIN {X 0,Y 333.806,Z 266.53,A -85,B 0,C 180,E1 -14575.169,E2 -14575.169} C_VEL
LIN {X 0,Y 334.102,Z 266.483,A -85,B 0,C 180,E1 -14577.589,E2 -14577.589} C_VEL
LIN {X 0,Y 334.242,Z 266.475,A -85,B 0,C 180,E1 -14580,E2 -14580} C_VEL
LIN {X 0,Y 334.102,Z 266.481,A -85,B 0,C 180,E1 -14582.412,E2 -14582.412} C_VEL
LIN {X 0,Y 334.02,Z 266.493,A -85,B 0,C 180,E1 -14587.253,E2 -14587.253} C_VEL
LIN {X 0,Y 333.829,Z 266.52,A -85,B 0,C 180,E1 -14590.923,E2 -14590.923} C_VEL
LIN {X 0,Y 333.804,Z 266.528,A -85,B 0,C 180,E1 -14594.635,E2 -14594.635} C_VEL
LIN {X 0,Y 333.792,Z 266.531,A -85,B 0,C 180,E1 -14598.655,E2 -14598.655} C_VEL
LIN {X 0,Y 333.689,Z 266.544,A -85,B 0,C 180,E1 -14602.279,E2 -14602.279} C_VEL
LIN {X 0,Y 333.732,Z 266.539,A -85,B 0,C 180,E1 -14606.247,E2 -14606.247} C_VEL
LIN {X 0,Y 333.687,Z 266.518,A -85,B 0,C 180,E1 -14608.975,E2 -14608.975} C_VEL
LIN {X 0,Y 333.641,Z 266.553,A -85,B 0,C 180,E1 -14612.588,E2 -14612.588} C_VEL
LIN {X 0,Y 333.676,Z 266.532,A -85,B 0,C 180,E1 -14616.14,E2 -14616.14} C_VEL
LIN {X 0,Y 333.646,Z 266.535,A -85,B 0,C 180,E1 -14619.193,E2 -14619.193} C_VEL
LIN {X 0,Y 333.632,Z 266.552,A -85,B 0,C 180,E1 -14622.501,E2 -14622.501} C_VEL
LIN {X 0,Y 333.597,Z 266.558,A -85,B 0,C 180,E1 -14625.956,E2 -14625.956} C_VEL
LIN {X 0,Y 333.648,Z 266.55,A -85,B 0,C 180,E1 -14629.316,E2 -14629.316} C_VEL
LIN {X 0,Y 333.683,Z 266.687,A -85,B 0,C 180,E1 -14630.874,E2 -14630.874} C_VEL
LIN {X 0,Y 336.826,Z 277.935,A -85,B 0,C 180,E1 -14634.252,E2 -14634.252} C_VEL
LIN {X 0,Y 339.535,Z 289.441,A -85,B 0,C 180,E1 -14637.441,E2 -14637.441} C_VEL
LIN {X 0,Y 341.64,Z 299.49,A -85,B 0,C 180,E1 -14640.071,E2 -14640.071} C_VEL
LIN {X 0,Y 340.757,Z 306.633,A -85,B 0,C 180,E1 -14641.682,E2 -14641.682} C_VEL
LIN {X 0,Y 340.202,Z 311.292,A -85,B 0,C 180,E1 -14642.68,E2 -14642.68} C_VEL
LIN {X 0,Y 345.895,Z 340.924,A -85,B 0,C 180,E1 -14643.847,E2 -14643.847} C_VEL
LIN {X 0,Y 347.243,Z 349.542,A -85,B 0,C 180,E1 -14644.141,E2 -14644.141} C_VEL
LIN {X 0,Y 345.578,Z 425.722,A -85,B 0,C 180,E1 -14645.641,E2 -14645.641} C_VEL
LIN {X 0,Y 344.812,Z 438.999,A -85,B 0,C 180,E1 -14646.103,E2 -14646.103} C_VEL
LIN {X 0,Y 343.916,Z 451.5,A -85,B 0,C 180,E1 -14646.78,E2 -14646.78} C_VEL
LIN {X 0,Y 342.683,Z 464.295,A -85,B 0,C 180,E1 -14647.729,E2 -14647.729} C_VEL
LIN {X 0,Y 341.189,Z 476.062,A -85,B 0,C 180,E1 -14648.871,E2 -14648.871} C_VEL
LIN {X 0,Y 339.558,Z 486.758,A -85,B 0,C 180,E1 -14650.189,E2 -14650.189} C_VEL
LIN {X 0,Y 338.179,Z 495.532,A -85,B 0,C 180,E1 -14651.523,E2 -14651.523} C_VEL
LIN {X 0,Y 336.491,Z 505.09,A -85,B 0,C 180,E1 -14653.311,E2 -14653.311} C_VEL
LIN {X 0,Y 335.231,Z 512.566,A -85,B 0,C 180,E1 -14655.059,E2 -14655.059} C_VEL
LIN {X 0,Y 334.392,Z 518.028,A -85,B 0,C 180,E1 -14656.633,E2 -14656.633} C_VEL
LIN {X 0,Y 333.444,Z 523.193,A -85,B 0,C 180,E1 -14658.45,E2 -14658.45} C_VEL
LIN {X 0,Y 332.864,Z 527.249,A -85,B 0,C 180,E1 -14660.276,E2 -14660.276} C_VEL
LIN {X 0,Y 332.588,Z 529.417,A -85,B 0,C 180,E1 -14661.494,E2 -14661.494} C_VEL
LIN {X 0,Y 332.342,Z 531.158,A -85,B 0,C 180,E1 -14662.711,E2 -14662.711} C_VEL
LIN {X 0,Y 332.096,Z 533.433,A -85,B 0,C 180,E1 -14665.144,E2 -14665.144} C_VEL
LIN {X 0,Y 331.957,Z 534.263,A -85,B 0,C 180,E1 -14667.573,E2 -14667.573} C_VEL
LIN {X 0,Y 331.954,Z 534.134,A -85,B 0,C 180,E1 -14668.787,E2 -14668.787} C_VEL
LIN {X 0,Y 332.04,Z 532.737,A -85,B 0,C 180,E1 -14671.213,E2 -14671.213} C_VEL
LIN {X 0,Y 332.355,Z 529.871,A -85,B 0,C 180,E1 -14673.637,E2 -14673.637} C_VEL
LIN {X 0,Y 332.743,Z 526.644,A -85,B 0,C 180,E1 -14675.454,E2 -14675.454} C_VEL
LIN {X 0,Y 333.297,Z 522.425,A -85,B 0,C 180,E1 -14677.268,E2 -14677.268} C_VEL
LIN {X 0,Y 334.13,Z 516.114,A -85,B 0,C 180,E1 -14679.381,E2 -14679.381} C_VEL
LIN {X 0,Y 335.154,Z 509.266,A -85,B 0,C 180,E1 -14681.184,E2 -14681.184} C_VEL
LIN {X 0,Y 336.469,Z 500.761,A -85,B 0,C 180,E1 -14682.976,E2 -14682.976} C_VEL
LIN {X 0,Y 337.738,Z 492.113,A -85,B 0,C 180,E1 -14684.46,E2 -14684.46} C_VEL
LIN {X 0,Y 339.03,Z 482.676,A -85,B 0,C 180,E1 -14685.788,E2 -14685.788} C_VEL
LIN {X 0,Y 340.4,Z 471.016,A -85,B 0,C 180,E1 -14687.11,E2 -14687.11} C_VEL
LIN {X 0,Y 341.725,Z 459.424,A -85,B 0,C 180,E1 -14688.123,E2 -14688.123} C_VEL
LIN {X 0,Y 342.794,Z 447.467,A -85,B 0,C 180,E1 -14688.916,E2 -14688.916} C_VEL
LIN {X 0,Y 343.573,Z 433.949,A -85,B 0,C 180,E1 -14689.557,E2 -14689.557} C_VEL
LIN {X 0,Y 344.082,Z 421.506,A -85,B 0,C 180,E1 -14689.918,E2 -14689.918} C_VEL
LIN {X 0,Y 345.419,Z 348.012,A -85,B 0,C 180,E1 -14691.359,E2 -14691.359} C_VEL
LIN {X 0,Y 341.386,Z 323.61,A -85,B 0,C 180,E1 -14692.179,E2 -14692.179} C_VEL
LIN {X 0,Y 340.059,Z 319.853,A -85,B 0,C 180,E1 -14692.363,E2 -14692.363} C_VEL
LIN {X 0,Y 337.978,Z 316.544,A -85,B 0,C 180,E1 -14692.614,E2 -14692.614} C_VEL
LIN {X 0,Y 334.445,Z 311.719,A -85,B 0,C 180,E1 -14693.201,E2 -14693.201} C_VEL
LIN {X 0,Y 333,Z 308.601,A -85,B 0,C 180,E1 -14693.753,E2 -14693.753} C_VEL
LIN {X 0,Y 332.936,Z 307.342,A -85,B 0,C 180,E1 -14694.021,E2 -14694.021} C_VEL
LIN {X 0,Y 333.981,Z 299.116,A -85,B 0,C 180,E1 -14695.889,E2 -14695.889} C_VEL
LIN {X 0,Y 331.839,Z 287.969,A -85,B 0,C 180,E1 -14698.804,E2 -14698.804} C_VEL
LIN {X 0,Y 328.734,Z 275.44,A -85,B 0,C 180,E1 -14702.308,E2 -14702.308} C_VEL
LIN {X 0,Y 326.647,Z 267.492,A -85,B 0,C 180,E1 -14704.714,E2 -14704.714} C_VEL
LIN {X 0,Y 326.598,Z 267.423,A -85,B 0,C 180,E1 -14708.611,E2 -14708.611} C_VEL
LIN {X 0,Y 326.576,Z 267.422,A -85,B 0,C 180,E1 -14711.845,E2 -14711.845} C_VEL
LIN {X 0,Y 326.527,Z 267.421,A -85,B 0,C 180,E1 -14715.256,E2 -14715.256} C_VEL
LIN {X 0,Y 326.576,Z 267.417,A -85,B 0,C 180,E1 -14718.868,E2 -14718.868} C_VEL
LIN {X 0,Y 326.626,Z 267.424,A -85,B 0,C 180,E1 -14722.76,E2 -14722.76} C_VEL
LIN {X 0,Y 326.604,Z 267.398,A -85,B 0,C 180,E1 -14725.98,E2 -14725.98} C_VEL
LIN {X 0,Y 326.658,Z 267.42,A -85,B 0,C 180,E1 -14730.34,E2 -14730.34} C_VEL
LIN {X 0,Y 326.686,Z 267.417,A -85,B 0,C 180,E1 -14734.515,E2 -14734.515} C_VEL
LIN {X 0,Y 326.642,Z 267.424,A -85,B 0,C 180,E1 -14738.544,E2 -14738.544} C_VEL
LIN {X 0,Y 326.74,Z 267.404,A -85,B 0,C 180,E1 -14741.177,E2 -14741.177} C_VEL
LIN {X 0,Y 326.758,Z 267.398,A -85,B 0,C 180,E1 -14745.432,E2 -14745.432} C_VEL
LIN {X 0,Y 326.764,Z 267.401,A -85,B 0,C 180,E1 -14748.838,E2 -14748.838} C_VEL
LIN {X 0,Y 326.953,Z 267.385,A -85,B 0,C 180,E1 -14752.589,E2 -14752.589} C_VEL
LIN {X 0,Y 326.771,Z 267.393,A -85,B 0,C 180,E1 -14755.064,E2 -14755.064} C_VEL
LIN {X 0,Y 327.042,Z 267.37,A -85,B 0,C 180,E1 -14757.536,E2 -14757.536} C_VEL
LIN {X 0,Y 327.192,Z 267.345,A -85,B 0,C 180,E1 -14760,E2 -14760} C_VEL
LIN {X 0,Y 327.042,Z 267.37,A -85,B 0,C 180,E1 -14762.463,E2 -14762.463} C_VEL
LIN {X 0,Y 326.99,Z 267.367,A -85,B 0,C 180,E1 -14766.169,E2 -14766.169} C_VEL
LIN {X 0,Y 326.909,Z 267.388,A -85,B 0,C 180,E1 -14768.655,E2 -14768.655} C_VEL
LIN {X 0,Y 326.728,Z 267.407,A -85,B 0,C 180,E1 -14772.421,E2 -14772.421} C_VEL
LIN {X 0,Y 326.748,Z 267.402,A -85,B 0,C 180,E1 -14774.957,E2 -14774.957} C_VEL
LIN {X 0,Y 326.727,Z 267.409,A -85,B 0,C 180,E1 -14778.838,E2 -14778.838} C_VEL
LIN {X 0,Y 326.615,Z 267.425,A -85,B 0,C 180,E1 -14782.787,E2 -14782.787} C_VEL
LIN {X 0,Y 326.685,Z 267.41,A -85,B 0,C 180,E1 -14785.484,E2 -14785.484} C_VEL
LIN {X 0,Y 326.656,Z 267.394,A -85,B 0,C 180,E1 -14789.659,E2 -14789.659} C_VEL
LIN {X 0,Y 326.603,Z 267.429,A -85,B 0,C 180,E1 -14794.02,E2 -14794.02} C_VEL
LIN {X 0,Y 326.623,Z 267.402,A -85,B 0,C 180,E1 -14797.239,E2 -14797.239} C_VEL
LIN {X 0,Y 326.573,Z 267.421,A -85,B 0,C 180,E1 -14801.132,E2 -14801.132} C_VEL
LIN {X 0,Y 326.553,Z 267.433,A -85,B 0,C 180,E1 -14804.748,E2 -14804.748} C_VEL
LIN {X 0,Y 326.573,Z 267.377,A -85,B 0,C 180,E1 -14808.155,E2 -14808.155} C_VEL
LIN {X 0,Y 326.62,Z 267.428,A -85,B 0,C 180,E1 -14811.392,E2 -14811.392} C_VEL
LIN {X 0,Y 326.676,Z 267.57,A -85,B 0,C 180,E1 -14813.705,E2 -14813.705} C_VEL
LIN {X 0,Y 330.007,Z 279.909,A -85,B 0,C 180,E1 -14817.108,E2 -14817.108} C_VEL
LIN {X 0,Y 333.222,Z 293.104,A -85,B 0,C 180,E1 -14820.478,E2 -14820.478} C_VEL
LIN {X 0,Y 334.679,Z 299.682,A -85,B 0,C 180,E1 -14822.021,E2 -14822.021} C_VEL
LIN {X 0,Y 335.887,Z 303.36,A -85,B 0,C 180,E1 -14822.239,E2 -14822.239} C_VEL
LIN {X 0,Y 339.921,Z 330.378,A -85,B 0,C 180,E1 -14823.204,E2 -14823.204} C_VEL
LIN {X 0,Y 337.27,Z 431.53,A -85,B 0,C 180,E1 -14825.453,E2 -14825.453} C_VEL
LIN {X 0,Y 336.39,Z 445.757,A -85,B 0,C 180,E1 -14826,E2 -14826} C_VEL
LIN {X 0,Y 335.315,Z 459.488,A -85,B 0,C 180,E1 -14826.778,E2 -14826.778} C_VEL
LIN {X 0,Y 334.025,Z 472.721,A -85,B 0,C 180,E1 -14827.785,E2 -14827.785} C_VEL
LIN {X 0,Y 332.67,Z 484.735,A -85,B 0,C 180,E1 -14828.953,E2 -14828.953} C_VEL
LIN {X 0,Y 331.039,Z 496.063,A -85,B 0,C 180,E1 -14830.305,E2 -14830.305} C_VEL
LIN {X 0,Y 329.508,Z 507.36,A -85,B 0,C 180,E1 -14831.985,E2 -14831.985} C_VEL
LIN {X 0,Y 328.135,Z 517.451,A -85,B 0,C 180,E1 -14833.834,E2 -14833.834} C_VEL
LIN {X 0,Y 327.211,Z 525.787,A -85,B 0,C 180,E1 -14835.7,E2 -14835.7} C_VEL
LIN {X 0,Y 326.167,Z 533.714,A -85,B 0,C 180,E1 -14837.873,E2 -14837.873} C_VEL
LIN {X 0,Y 325.456,Z 540.031,A -85,B 0,C 180,E1 -14840.052,E2 -14840.052} C_VEL
LIN {X 0,Y 325.143,Z 544.299,A -85,B 0,C 180,E1 -14841.924,E2 -14841.924} C_VEL
LIN {X 0,Y 324.881,Z 548.434,A -85,B 0,C 180,E1 -14844.322,E2 -14844.322} C_VEL
LIN {X 0,Y 324.862,Z 550.737,A -85,B 0,C 180,E1 -14846.279,E2 -14846.279} C_VEL
LIN {X 0,Y 324.83,Z 552.364,A -85,B 0,C 180,E1 -14848.76,E2 -14848.76} C_VEL
LIN {X 0,Y 324.873,Z 552.643,A -85,B 0,C 180,E1 -14850,E2 -14850} C_VEL
LIN {X 0,Y 324.83,Z 552.128,A -85,B 0,C 180,E1 -14852.48,E2 -14852.48} C_VEL
LIN {X 0,Y 324.865,Z 551.337,A -85,B 0,C 180,E1 -14853.721,E2 -14853.721} C_VEL
LIN {X 0,Y 324.956,Z 548.635,A -85,B 0,C 180,E1 -14856.208,E2 -14856.208} C_VEL
LIN {X 0,Y 325.268,Z 544.4,A -85,B 0,C 180,E1 -14858.699,E2 -14858.699} C_VEL
LIN {X 0,Y 325.854,Z 538.528,A -85,B 0,C 180,E1 -14861.193,E2 -14861.193} C_VEL
LIN {X 0,Y 326.838,Z 531.879,A -85,B 0,C 180,E1 -14863.365,E2 -14863.365} C_VEL
LIN {X 0,Y 328.008,Z 523.617,A -85,B 0,C 180,E1 -14865.522,E2 -14865.522} C_VEL
LIN {X 0,Y 329.322,Z 514.799,A -85,B 0,C 180,E1 -14867.384,E2 -14867.384} C_VEL
LIN {X 0,Y 330.966,Z 504.138,A -85,B 0,C 180,E1 -14869.216,E2 -14869.216} C_VEL
LIN {X 0,Y 332.67,Z 493.344,A -85,B 0,C 180,E1 -14870.723,E2 -14870.723} C_VEL
LIN {X 0,Y 334.307,Z 481.502,A -85,B 0,C 180,E1 -14872.072,E2 -14872.072} C_VEL
LIN {X 0,Y 335.664,Z 470.295,A -85,B 0,C 180,E1 -14873.101,E2 -14873.101} C_VEL
LIN {X 0,Y 336.966,Z 457.959,A -85,B 0,C 180,E1 -14873.998,E2 -14873.998} C_VEL
LIN {X 0,Y 338.183,Z 443.799,A -85,B 0,C 180,E1 -14874.763,E2 -14874.763} C_VEL
LIN {X 0,Y 339.028,Z 429.592,A -85,B 0,C 180,E1 -14875.271,E2 -14875.271} C_VEL
LIN {X 0,Y 341.73,Z 331.804,A -85,B 0,C 180,E1 -14877.434,E2 -14877.434} C_VEL
LIN {X 0,Y 340.255,Z 320.681,A -85,B 0,C 180,E1 -14877.832,E2 -14877.832} C_VEL
LIN {X 0,Y 337.568,Z 305.624,A -85,B 0,C 180,E1 -14878.44,E2 -14878.44} C_VEL
LIN {X 0,Y 335.049,Z 299.568,A -85,B 0,C 180,E1 -14878.866,E2 -14878.866} C_VEL
LIN {X 0,Y 332.177,Z 287.445,A -85,B 0,C 180,E1 -14881.933,E2 -14881.933} C_VEL
LIN {X 0,Y 329.438,Z 277.05,A -85,B 0,C 180,E1 -14884.77,E2 -14884.77} C_VEL
LIN {X 0,Y 326.637,Z 267.505,A -85,B 0,C 180,E1 -14887.584,E2 -14887.584} C_VEL
LIN {X 0,Y 326.626,Z 267.414,A -85,B 0,C 180,E1 -14891.141,E2 -14891.141} C_VEL
LIN {X 0,Y 326.588,Z 267.415,A -85,B 0,C 180,E1 -14894.754,E2 -14894.754} C_VEL
LIN {X 0,Y 326.573,Z 267.414,A -85,B 0,C 180,E1 -14898.154,E2 -14898.154} C_VEL
LIN {X 0,Y 326.62,Z 267.426,A -85,B 0,C 180,E1 -14901.391,E2 -14901.391} C_VEL
LIN {X 0,Y 326.615,Z 267.406,A -85,B 0,C 180,E1 -14904.851,E2 -14904.851} C_VEL
LIN {X 0,Y 326.603,Z 267.428,A -85,B 0,C 180,E1 -14907.455,E2 -14907.455} C_VEL
LIN {X 0,Y 326.656,Z 267.39,A -85,B 0,C 180,E1 -14910.341,E2 -14910.341} C_VEL
LIN {X 0,Y 326.685,Z 267.413,A -85,B 0,C 180,E1 -14914.516,E2 -14914.516} C_VEL
LIN {X 0,Y 326.642,Z 267.417,A -85,B 0,C 180,E1 -14918.545,E2 -14918.545} C_VEL
LIN {X 0,Y 326.74,Z 267.408,A -85,B 0,C 180,E1 -14921.178,E2 -14921.178} C_VEL
LIN {X 0,Y 326.758,Z 267.405,A -85,B 0,C 180,E1 -14925.433,E2 -14925.433} C_VEL
LIN {X 0,Y 326.764,Z 267.398,A -85,B 0,C 180,E1 -14928.839,E2 -14928.839} C_VEL
LIN {X 0,Y 326.961,Z 267.369,A -85,B 0,C 180,E1 -14932.59,E2 -14932.59} C_VEL
LIN {X 0,Y 326.772,Z 267.405,A -85,B 0,C 180,E1 -14935.065,E2 -14935.065} C_VEL
LIN {X 0,Y 327.042,Z 267.362,A -85,B 0,C 180,E1 -14937.537,E2 -14937.537} C_VEL
LIN {X 0,Y 327.193,Z 267.353,A -85,B 0,C 180,E1 -14940,E2 -14940} C_VEL
LIN {X 0,Y 327.043,Z 267.36,A -85,B 0,C 180,E1 -14942.464,E2 -14942.464} C_VEL
LIN {X 0,Y 326.966,Z 267.371,A -85,B 0,C 180,E1 -14946.671,E2 -14946.671} C_VEL
LIN {X 0,Y 326.809,Z 267.398,A -85,B 0,C 180,E1 -14949.907,E2 -14949.907} C_VEL
LIN {X 0,Y 326.755,Z 267.408,A -85,B 0,C 180,E1 -14953.686,E2 -14953.686} C_VEL
LIN {X 0,Y 326.696,Z 267.417,A -85,B 0,C 180,E1 -14957.529,E2 -14957.529} C_VEL
LIN {X 0,Y 326.659,Z 267.411,A -85,B 0,C 180,E1 -14960.136,E2 -14960.136} C_VEL
LIN {X 0,Y 326.649,Z 267.414,A -85,B 0,C 180,E1 -14964.13,E2 -14964.13} C_VEL
LIN {X 0,Y 326.68,Z 267.411,A -85,B 0,C 180,E1 -14966.859,E2 -14966.859} C_VEL
LIN {X 0,Y 326.632,Z 267.411,A -85,B 0,C 180,E1 -14970.61,E2 -14970.61} C_VEL
LIN {X 0,Y 326.605,Z 267.411,A -85,B 0,C 180,E1 -14974.02,E2 -14974.02} C_VEL
LIN {X 0,Y 326.628,Z 267.424,A -85,B 0,C 180,E1 -14977.24,E2 -14977.24} C_VEL
LIN {X 0,Y 326.577,Z 267.419,A -85,B 0,C 180,E1 -14981.132,E2 -14981.132} C_VEL
LIN {X 0,Y 326.527,Z 267.425,A -85,B 0,C 180,E1 -14984.744,E2 -14984.744} C_VEL
LIN {X 0,Y 326.577,Z 267.421,A -85,B 0,C 180,E1 -14988.155,E2 -14988.155} C_VEL
LIN {X 0,Y 326.621,Z 267.6,A -85,B 0,C 180,E1 -14990.166,E2 -14990.166} C_VEL
LIN {X 0,Y 329.648,Z 278.358,A -85,B 0,C 180,E1 -14993.499,E2 -14993.499} C_VEL
LIN {X 0,Y 331.838,Z 287.166,A -85,B 0,C 180,E1 -14996.047,E2 -14996.047} C_VEL
LIN {X 0,Y 334.596,Z 299.692,A -85,B 0,C 180,E1 -14999.451,E2 -14999.451} C_VEL
LIN {X 0,Y 334.84,Z 302.26,A -85,B 0,C 180,E1 -15000.1,E2 -15000.1} C_VEL
LIN {X 0,Y 333.599,Z 311.132,A -85,B 0,C 180,E1 -15002.08,E2 -15002.08} C_VEL
LIN {X 0,Y 338.537,Z 336.619,A -85,B 0,C 180,E1 -15003.131,E2 -15003.131} C_VEL
LIN {X 0,Y 340.865,Z 350.238,A -85,B 0,C 180,E1 -15003.629,E2 -15003.629} C_VEL
LIN {X 0,Y 339.167,Z 424.31,A -85,B 0,C 180,E1 -15005.109,E2 -15005.109} C_VEL
LIN {X 0,Y 338.507,Z 437.493,A -85,B 0,C 180,E1 -15005.548,E2 -15005.548} C_VEL
LIN {X 0,Y 337.52,Z 450.349,A -85,B 0,C 180,E1 -15006.224,E2 -15006.224} C_VEL
LIN {X 0,Y 336.242,Z 463.217,A -85,B 0,C 180,E1 -15007.171,E2 -15007.171} C_VEL
LIN {X 0,Y 334.74,Z 474.809,A -85,B 0,C 180,E1 -15008.282,E2 -15008.282} C_VEL
LIN {X 0,Y 333.082,Z 485.805,A -85,B 0,C 180,E1 -15009.626,E2 -15009.626} C_VEL
LIN {X 0,Y 331.433,Z 495.645,A -85,B 0,C 180,E1 -15011.133,E2 -15011.133} C_VEL
LIN {X 0,Y 329.677,Z 505.211,A -85,B 0,C 180,E1 -15012.955,E2 -15012.955} C_VEL
LIN {X 0,Y 328.304,Z 512.908,A -85,B 0,C 180,E1 -15014.793,E2 -15014.793} C_VEL
LIN {X 0,Y 327.467,Z 518.167,A -85,B 0,C 180,E1 -15016.345,E2 -15016.345} C_VEL
LIN {X 0,Y 326.443,Z 523.341,A -85,B 0,C 180,E1 -15018.198,E2 -15018.198} C_VEL
LIN {X 0,Y 325.836,Z 527.408,A -85,B 0,C 180,E1 -15020.064,E2 -15020.064} C_VEL
LIN {X 0,Y 325.557,Z 529.58,A -85,B 0,C 180,E1 -15021.309,E2 -15021.309} C_VEL
LIN {X 0,Y 325.286,Z 531.331,A -85,B 0,C 180,E1 -15022.552,E2 -15022.552} C_VEL
LIN {X 0,Y 325.001,Z 533.618,A -85,B 0,C 180,E1 -15025.038,E2 -15025.038} C_VEL
LIN {X 0,Y 324.964,Z 534.215,A -85,B 0,C 180,E1 -15026.28,E2 -15026.28} C_VEL
LIN {X 0,Y 324.862,Z 534.34,A -85,B 0,C 180,E1 -15028.76,E2 -15028.76} C_VEL
LIN {X 0,Y 324.946,Z 532.959,A -85,B 0,C 180,E1 -15031.239,E2 -15031.239} C_VEL
LIN {X 0,Y 325.284,Z 530.107,A -85,B 0,C 180,E1 -15033.716,E2 -15033.716} C_VEL
LIN {X 0,Y 325.703,Z 526.896,A -85,B 0,C 180,E1 -15035.572,E2 -15035.572} C_VEL
LIN {X 0,Y 326.265,Z 522.695,A -85,B 0,C 180,E1 -15037.426,E2 -15037.426} C_VEL
LIN {X 0,Y 327.149,Z 516.406,A -85,B 0,C 180,E1 -15039.584,E2 -15039.584} C_VEL
LIN {X 0,Y 328.201,Z 509.592,A -85,B 0,C 180,E1 -15041.424,E2 -15041.424} C_VEL
LIN {X 0,Y 329.561,Z 501.128,A -85,B 0,C 180,E1 -15043.252,E2 -15043.252} C_VEL
LIN {X 0,Y 330.889,Z 492.523,A -85,B 0,C 180,E1 -15044.766,E2 -15044.766} C_VEL
LIN {X 0,Y 332.238,Z 483.141,A -85,B 0,C 180,E1 -15046.119,E2 -15046.119} C_VEL
LIN {X 0,Y 333.653,Z 471.554,A -85,B 0,C 180,E1 -15047.467,E2 -15047.467} C_VEL
LIN {X 0,Y 335.026,Z 460.113,A -85,B 0,C 180,E1 -15048.498,E2 -15048.498} C_VEL
LIN {X 0,Y 336.129,Z 448.379,A -85,B 0,C 180,E1 -15049.306,E2 -15049.306} C_VEL
LIN {X 0,Y 336.937,Z 435.084,A -85,B 0,C 180,E1 -15049.964,E2 -15049.964} C_VEL
LIN {X 0,Y 337.516,Z 422.288,A -85,B 0,C 180,E1 -15050.356,E2 -15050.356} C_VEL
LIN {X 0,Y 338.89,Z 348.523,A -85,B 0,C 180,E1 -15051.837,E2 -15051.837} C_VEL
LIN {X 0,Y 333.93,Z 319.15,A -85,B 0,C 180,E1 -15052.866,E2 -15052.866} C_VEL
LIN {X 0,Y 332.47,Z 311.261,A -85,B 0,C 180,E1 -15053.194,E2 -15053.194} C_VEL
LIN {X 0,Y 332.936,Z 307.342,A -85,B 0,C 180,E1 -15054.021,E2 -15054.021} C_VEL
LIN {X 0,Y 332.626,Z 303.956,A -85,B 0,C 180,E1 -15054.851,E2 -15054.851} C_VEL
LIN {X 0,Y 331.183,Z 300.931,A -85,B 0,C 180,E1 -15055.7,E2 -15055.7} C_VEL
LIN {X 0,Y 326.045,Z 293.39,A -85,B 0,C 180,E1 -15058.028,E2 -15058.028} C_VEL
LIN {X 0,Y 325.353,Z 291.281,A -85,B 0,C 180,E1 -15058.623,E2 -15058.623} C_VEL
LIN {X 0,Y 322.644,Z 279.907,A -85,B 0,C 180,E1 -15061.839,E2 -15061.839} C_VEL
LIN {X 0,Y 319.607,Z 268.39,A -85,B 0,C 180,E1 -15065.35,E2 -15065.35} C_VEL
LIN {X 0,Y 319.544,Z 268.298,A -85,B 0,C 180,E1 -15068.011,E2 -15068.011} C_VEL
LIN {X 0,Y 319.526,Z 268.298,A -85,B 0,C 180,E1 -15071.596,E2 -15071.596} C_VEL
LIN {X 0,Y 319.487,Z 268.297,A -85,B 0,C 180,E1 -15075.256,E2 -15075.256} C_VEL
LIN {X 0,Y 319.527,Z 268.297,A -85,B 0,C 180,E1 -15078.711,E2 -15078.711} C_VEL
LIN {X 0,Y 319.575,Z 268.3,A -85,B 0,C 180,E1 -15082.343,E2 -15082.343} C_VEL
LIN {X 0,Y 319.558,Z 268.283,A -85,B 0,C 180,E1 -15085.122,E2 -15085.122} C_VEL
LIN {X 0,Y 319.568,Z 268.301,A -85,B 0,C 180,E1 -15089.057,E2 -15089.057} C_VEL
LIN {X 0,Y 319.606,Z 268.292,A -85,B 0,C 180,E1 -15092.497,E2 -15092.497} C_VEL
LIN {X 0,Y 319.6,Z 268.29,A -85,B 0,C 180,E1 -15095.303,E2 -15095.303} C_VEL
LIN {X 0,Y 319.593,Z 268.299,A -85,B 0,C 180,E1 -15098.047,E2 -15098.047} C_VEL
LIN {X 0,Y 319.685,Z 268.281,A -85,B 0,C 180,E1 -15100.962,E2 -15100.962} C_VEL
LIN {X 0,Y 319.726,Z 268.273,A -85,B 0,C 180,E1 -15105.275,E2 -15105.275} C_VEL
LIN {X 0,Y 319.747,Z 268.269,A -85,B 0,C 180,E1 -15109.872,E2 -15109.872} C_VEL
LIN {X 0,Y 319.907,Z 268.261,A -85,B 0,C 180,E1 -15112.425,E2 -15112.425} C_VEL
LIN {X 0,Y 319.74,Z 268.269,A -85,B 0,C 180,E1 -15114.956,E2 -15114.956} C_VEL
LIN {X 0,Y 319.986,Z 268.249,A -85,B 0,C 180,E1 -15117.482,E2 -15117.482} C_VEL
LIN {X 0,Y 320.144,Z 268.222,A -85,B 0,C 180,E1 -15120,E2 -15120} C_VEL
LIN {X 0,Y 319.986,Z 268.249,A -85,B 0,C 180,E1 -15122.517,E2 -15122.517} C_VEL
LIN {X 0,Y 319.946,Z 268.244,A -85,B 0,C 180,E1 -15126.305,E2 -15126.305} C_VEL
LIN {X 0,Y 319.837,Z 268.268,A -85,B 0,C 180,E1 -15128.848,E2 -15128.848} C_VEL
LIN {X 0,Y 319.676,Z 268.29,A -85,B 0,C 180,E1 -15132.7,E2 -15132.7} C_VEL
LIN {X 0,Y 319.694,Z 268.28,A -85,B 0,C 180,E1 -15135.295,E2 -15135.295} C_VEL
LIN {X 0,Y 319.669,Z 268.288,A -85,B 0,C 180,E1 -15139.255,E2 -15139.255} C_VEL
LIN {X 0,Y 319.565,Z 268.303,A -85,B 0,C 180,E1 -15143.319,E2 -15143.319} C_VEL
LIN {X 0,Y 319.63,Z 268.294,A -85,B 0,C 180,E1 -15146.088,E2 -15146.088} C_VEL
LIN {X 0,Y 319.585,Z 268.283,A -85,B 0,C 180,E1 -15148.934,E2 -15148.934} C_VEL
LIN {X 0,Y 319.528,Z 268.29,A -85,B 0,C 180,E1 -15151.862,E2 -15151.862} C_VEL
LIN {X 0,Y 319.575,Z 268.288,A -85,B 0,C 180,E1 -15155.543,E2 -15155.543} C_VEL
LIN {X 0,Y 319.553,Z 268.29,A -85,B 0,C 180,E1 -15158.011,E2 -15158.011} C_VEL
LIN {X 0,Y 319.521,Z 268.294,A -85,B 0,C 180,E1 -15161.597,E2 -15161.597} C_VEL
LIN {X 0,Y 319.512,Z 268.302,A -85,B 0,C 180,E1 -15165.263,E2 -15165.263} C_VEL
LIN {X 0,Y 319.524,Z 268.255,A -85,B 0,C 180,E1 -15168.712,E2 -15168.712} C_VEL
LIN {X 0,Y 319.589,Z 268.3,A -85,B 0,C 180,E1 -15172.79,E2 -15172.79} C_VEL
LIN {X 0,Y 319.654,Z 268.635,A -85,B 0,C 180,E1 -15173.095,E2 -15173.095} C_VEL
LIN {X 0,Y 322.936,Z 280.546,A -85,B 0,C 180,E1 -15176.474,E2 -15176.474} C_VEL
LIN {X 0,Y 325.861,Z 292.44,A -85,B 0,C 180,E1 -15179.621,E2 -15179.621} C_VEL
LIN {X 0,Y 327.526,Z 299.83,A -85,B 0,C 180,E1 -15181.419,E2 -15181.419} C_VEL
LIN {X 0,Y 329.737,Z 305.814,A -85,B 0,C 180,E1 -15181.788,E2 -15181.788} C_VEL
LIN {X 0,Y 333.438,Z 331.596,A -85,B 0,C 180,E1 -15182.723,E2 -15182.723} C_VEL
LIN {X 0,Y 330.744,Z 431.289,A -85,B 0,C 180,E1 -15184.977,E2 -15184.977} C_VEL
LIN {X 0,Y 329.844,Z 445.577,A -85,B 0,C 180,E1 -15185.534,E2 -15185.534} C_VEL
LIN {X 0,Y 328.775,Z 458.768,A -85,B 0,C 180,E1 -15186.288,E2 -15186.288} C_VEL
LIN {X 0,Y 327.443,Z 471.704,A -85,B 0,C 180,E1 -15187.274,E2 -15187.274} C_VEL
LIN {X 0,Y 326.015,Z 484.239,A -85,B 0,C 180,E1 -15188.502,E2 -15188.502} C_VEL
LIN {X 0,Y 324.348,Z 495.635,A -85,B 0,C 180,E1 -15189.881,E2 -15189.881} C_VEL
LIN {X 0,Y 323,Z 505.089,A -85,B 0,C 180,E1 -15191.281,E2 -15191.281} C_VEL
LIN {X 0,Y 321.689,Z 513.963,A -85,B 0,C 180,E1 -15192.847,E2 -15192.847} C_VEL
LIN {X 0,Y 320.475,Z 523.03,A -85,B 0,C 180,E1 -15194.778,E2 -15194.778} C_VEL
LIN {X 0,Y 319.465,Z 531.368,A -85,B 0,C 180,E1 -15196.968,E2 -15196.968} C_VEL
LIN {X 0,Y 318.568,Z 538.111,A -85,B 0,C 180,E1 -15199.192,E2 -15199.192} C_VEL
LIN {X 0,Y 318.176,Z 542.763,A -85,B 0,C 180,E1 -15201.106,E2 -15201.106} C_VEL
LIN {X 0,Y 317.878,Z 547.418,A -85,B 0,C 180,E1 -15203.653,E2 -15203.653} C_VEL
LIN {X 0,Y 317.771,Z 550.519,A -85,B 0,C 180,E1 -15206.196,E2 -15206.196} C_VEL
LIN {X 0,Y 317.741,Z 552.158,A -85,B 0,C 180,E1 -15208.733,E2 -15208.733} C_VEL
LIN {X 0,Y 317.78,Z 552.442,A -85,B 0,C 180,E1 -15210,E2 -15210} C_VEL
LIN {X 0,Y 317.751,Z 551.936,A -85,B 0,C 180,E1 -15212.535,E2 -15212.535} C_VEL
LIN {X 0,Y 317.775,Z 551.15,A -85,B 0,C 180,E1 -15213.804,E2 -15213.804} C_VEL
LIN {X 0,Y 317.882,Z 548.459,A -85,B 0,C 180,E1 -15216.347,E2 -15216.347} C_VEL
LIN {X 0,Y 318.201,Z 544.231,A -85,B 0,C 180,E1 -15218.894,E2 -15218.894} C_VEL
LIN {X 0,Y 318.843,Z 538.366,A -85,B 0,C 180,E1 -15221.442,E2 -15221.442} C_VEL
LIN {X 0,Y 319.862,Z 531.722,A -85,B 0,C 180,E1 -15223.662,E2 -15223.662} C_VEL
LIN {X 0,Y 321.127,Z 523.413,A -85,B 0,C 180,E1 -15225.876,E2 -15225.876} C_VEL
LIN {X 0,Y 322.493,Z 514.652,A -85,B 0,C 180,E1 -15227.764,E2 -15227.764} C_VEL
LIN {X 0,Y 324.236,Z 503.994,A -85,B 0,C 180,E1 -15229.631,E2 -15229.631} C_VEL
LIN {X 0,Y 326.021,Z 493.199,A -85,B 0,C 180,E1 -15231.166,E2 -15231.166} C_VEL
LIN {X 0,Y 327.71,Z 481.354,A -85,B 0,C 180,E1 -15232.541,E2 -15232.541} C_VEL
LIN {X 0,Y 329.168,Z 469.996,A -85,B 0,C 180,E1 -15233.598,E2 -15233.598} C_VEL
LIN {X 0,Y 330.464,Z 457.786,A -85,B 0,C 180,E1 -15234.5,E2 -15234.5} C_VEL
LIN {X 0,Y 331.76,Z 443.585,A -85,B 0,C 180,E1 -15235.276,E2 -15235.276} C_VEL
LIN {X 0,Y 332.634,Z 429.249,A -85,B 0,C 180,E1 -15235.792,E2 -15235.792} C_VEL
LIN {X 0,Y 335.42,Z 332.088,A -85,B 0,C 180,E1 -15237.976,E2 -15237.976} C_VEL
LIN {X 0,Y 331.795,Z 308.862,A -85,B 0,C 180,E1 -15238.888,E2 -15238.888} C_VEL
LIN {X 0,Y 327.924,Z 299.748,A -85,B 0,C 180,E1 -15239.533,E2 -15239.533} C_VEL
LIN {X 0,Y 324.963,Z 287.528,A -85,B 0,C 180,E1 -15242.729,E2 -15242.729} C_VEL
LIN {X 0,Y 322.172,Z 277.182,A -85,B 0,C 180,E1 -15245.668,E2 -15245.668} C_VEL
LIN {X 0,Y 319.609,Z 268.35,A -85,B 0,C 180,E1 -15248.403,E2 -15248.403} C_VEL
LIN {X 0,Y 319.593,Z 268.292,A -85,B 0,C 180,E1 -15251.611,E2 -15251.611} C_VEL
LIN {X 0,Y 319.561,Z 268.293,A -85,B 0,C 180,E1 -15255.27,E2 -15255.27} C_VEL
LIN {X 0,Y 319.525,Z 268.289,A -85,B 0,C 180,E1 -15258.711,E2 -15258.711} C_VEL
LIN {X 0,Y 319.573,Z 268.294,A -85,B 0,C 180,E1 -15262.344,E2 -15262.344} C_VEL
LIN {X 0,Y 319.555,Z 268.288,A -85,B 0,C 180,E1 -15265.123,E2 -15265.123} C_VEL
LIN {X 0,Y 319.566,Z 268.28,A -85,B 0,C 180,E1 -15269.058,E2 -15269.058} C_VEL
LIN {X 0,Y 319.605,Z 268.292,A -85,B 0,C 180,E1 -15272.498,E2 -15272.498} C_VEL
LIN {X 0,Y 319.6,Z 268.292,A -85,B 0,C 180,E1 -15275.304,E2 -15275.304} C_VEL
LIN {X 0,Y 319.592,Z 268.299,A -85,B 0,C 180,E1 -15278.048,E2 -15278.048} C_VEL
LIN {X 0,Y 319.684,Z 268.286,A -85,B 0,C 180,E1 -15280.962,E2 -15280.962} C_VEL
LIN {X 0,Y 319.726,Z 268.28,A -85,B 0,C 180,E1 -15285.276,E2 -15285.276} C_VEL
LIN {X 0,Y 319.752,Z 268.28,A -85,B 0,C 180,E1 -15289.873,E2 -15289.873} C_VEL
LIN {X 0,Y 319.92,Z 268.247,A -85,B 0,C 180,E1 -15292.426,E2 -15292.426} C_VEL
LIN {X 0,Y 319.742,Z 268.281,A -85,B 0,C 180,E1 -15294.956,E2 -15294.956} C_VEL
LIN {X 0,Y 319.986,Z 268.241,A -85,B 0,C 180,E1 -15297.483,E2 -15297.483} C_VEL
LIN {X 0,Y 320.145,Z 268.231,A -85,B 0,C 180,E1 -15300,E2 -15300} C_VEL
LIN {X 0,Y 319.987,Z 268.239,A -85,B 0,C 180,E1 -15302.518,E2 -15302.518} C_VEL
LIN {X 0,Y 319.926,Z 268.248,A -85,B 0,C 180,E1 -15306.662,E2 -15306.662} C_VEL
LIN {X 0,Y 319.753,Z 268.276,A -85,B 0,C 180,E1 -15310.128,E2 -15310.128} C_VEL
LIN {X 0,Y 319.727,Z 268.281,A -85,B 0,C 180,E1 -15314.725,E2 -15314.725} C_VEL
LIN {X 0,Y 319.686,Z 268.284,A -85,B 0,C 180,E1 -15319.038,E2 -15319.038} C_VEL
LIN {X 0,Y 319.567,Z 268.297,A -85,B 0,C 180,E1 -15323.32,E2 -15323.32} C_VEL
LIN {X 0,Y 319.631,Z 268.295,A -85,B 0,C 180,E1 -15326.089,E2 -15326.089} C_VEL
LIN {X 0,Y 319.577,Z 268.274,A -85,B 0,C 180,E1 -15328.935,E2 -15328.935} C_VEL
LIN {X 0,Y 319.528,Z 268.309,A -85,B 0,C 180,E1 -15331.863,E2 -15331.863} C_VEL
LIN {X 0,Y 319.578,Z 268.281,A -85,B 0,C 180,E1 -15335.544,E2 -15335.544} C_VEL
LIN {X 0,Y 319.573,Z 268.303,A -85,B 0,C 180,E1 -15338.009,E2 -15338.009} C_VEL
LIN {X 0,Y 319.525,Z 268.305,A -85,B 0,C 180,E1 -15341.598,E2 -15341.598} C_VEL
LIN {X 0,Y 319.488,Z 268.307,A -85,B 0,C 180,E1 -15345.258,E2 -15345.258} C_VEL
LIN {X 0,Y 319.529,Z 268.305,A -85,B 0,C 180,E1 -15348.713,E2 -15348.713} C_VEL
LIN {X 0,Y 319.578,Z 268.435,A -85,B 0,C 180,E1 -15349.386,E2 -15349.386} C_VEL
LIN {X 0,Y 322.571,Z 278.969,A -85,B 0,C 180,E1 -15352.773,E2 -15352.773} C_VEL
LIN {X 0,Y 324.743,Z 287.508,A -85,B 0,C 180,E1 -15355.325,E2 -15355.325} C_VEL
LIN {X 0,Y 327.711,Z 300.926,A -85,B 0,C 180,E1 -15359.075,E2 -15359.075} C_VEL
LIN {X 0,Y 328.076,Z 303.581,A -85,B 0,C 180,E1 -15359.774,E2 -15359.774} C_VEL
LIN {X 0,Y 327.043,Z 311.125,A -85,B 0,C 180,E1 -15361.473,E2 -15361.473} C_VEL
LIN {X 0,Y 332.305,Z 338.039,A -85,B 0,C 180,E1 -15362.611,E2 -15362.611} C_VEL
LIN {X 0,Y 334.52,Z 350.941,A -85,B 0,C 180,E1 -15363.099,E2 -15363.099} C_VEL
LIN {X 0,Y 332.81,Z 422.899,A -85,B 0,C 180,E1 -15364.558,E2 -15364.558} C_VEL
LIN {X 0,Y 332.123,Z 436.676,A -85,B 0,C 180,E1 -15365.004,E2 -15365.004} C_VEL
LIN {X 0,Y 331.179,Z 449.176,A -85,B 0,C 180,E1 -15365.648,E2 -15365.648} C_VEL
LIN {X 0,Y 330.007,Z 461.034,A -85,B 0,C 180,E1 -15366.5,E2 -15366.5} C_VEL
LIN {X 0,Y 328.375,Z 473.487,A -85,B 0,C 180,E1 -15367.673,E2 -15367.673} C_VEL
LIN {X 0,Y 326.586,Z 484.811,A -85,B 0,C 180,E1 -15369.037,E2 -15369.037} C_VEL
LIN {X 0,Y 324.981,Z 493.978,A -85,B 0,C 180,E1 -15370.416,E2 -15370.416} C_VEL
LIN {X 0,Y 323.428,Z 502.4,A -85,B 0,C 180,E1 -15371.962,E2 -15371.962} C_VEL
LIN {X 0,Y 321.806,Z 511.017,A -85,B 0,C 180,E1 -15373.933,E2 -15373.933} C_VEL
LIN {X 0,Y 320.553,Z 518.305,A -85,B 0,C 180,E1 -15376.045,E2 -15376.045} C_VEL
LIN {X 0,Y 319.462,Z 523.489,A -85,B 0,C 180,E1 -15377.937,E2 -15377.937} C_VEL
LIN {X 0,Y 318.821,Z 527.566,A -85,B 0,C 180,E1 -15379.843,E2 -15379.843} C_VEL
LIN {X 0,Y 318.511,Z 529.744,A -85,B 0,C 180,E1 -15381.115,E2 -15381.115} C_VEL
LIN {X 0,Y 318.224,Z 531.504,A -85,B 0,C 180,E1 -15382.385,E2 -15382.385} C_VEL
LIN {X 0,Y 317.911,Z 533.803,A -85,B 0,C 180,E1 -15384.927,E2 -15384.927} C_VEL
LIN {X 0,Y 317.894,Z 534.404,A -85,B 0,C 180,E1 -15386.197,E2 -15386.197} C_VEL
LIN {X 0,Y 317.772,Z 534.544,A -85,B 0,C 180,E1 -15388.733,E2 -15388.733} C_VEL
LIN {X 0,Y 317.856,Z 533.18,A -85,B 0,C 180,E1 -15391.267,E2 -15391.267} C_VEL
LIN {X 0,Y 318.215,Z 530.342,A -85,B 0,C 180,E1 -15393.799,E2 -15393.799} C_VEL
LIN {X 0,Y 318.663,Z 527.147,A -85,B 0,C 180,E1 -15395.696,E2 -15395.696} C_VEL
LIN {X 0,Y 319.374,Z 521.941,A -85,B 0,C 180,E1 -15398.002,E2 -15398.002} C_VEL
LIN {X 0,Y 320.31,Z 515.662,A -85,B 0,C 180,E1 -15400.109,E2 -15400.109} C_VEL
LIN {X 0,Y 321.493,Z 508.608,A -85,B 0,C 180,E1 -15401.986,E2 -15401.986} C_VEL
LIN {X 0,Y 322.953,Z 499.896,A -85,B 0,C 180,E1 -15403.85,E2 -15403.85} C_VEL
LIN {X 0,Y 324.297,Z 491.014,A -85,B 0,C 180,E1 -15405.395,E2 -15405.395} C_VEL
LIN {X 0,Y 325.777,Z 481.286,A -85,B 0,C 180,E1 -15406.77,E2 -15406.77} C_VEL
LIN {X 0,Y 327.11,Z 470.669,A -85,B 0,C 180,E1 -15407.989,E2 -15407.989} C_VEL
LIN {X 0,Y 328.524,Z 458.866,A -85,B 0,C 180,E1 -15409.04,E2 -15409.04} C_VEL
LIN {X 0,Y 329.692,Z 446.674,A -85,B 0,C 180,E1 -15409.86,E2 -15409.86} C_VEL
LIN {X 0,Y 330.448,Z 434.185,A -85,B 0,C 180,E1 -15410.468,E2 -15410.468} C_VEL
LIN {X 0,Y 331.031,Z 421.043,A -85,B 0,C 180,E1 -15410.86,E2 -15410.86} C_VEL
LIN {X 0,Y 332.402,Z 349.247,A -85,B 0,C 180,E1 -15412.327,E2 -15412.327} C_VEL
LIN {X 0,Y 327.663,Z 320.985,A -85,B 0,C 180,E1 -15413.345,E2 -15413.345} C_VEL
LIN {X 0,Y 325.829,Z 310.979,A -85,B 0,C 180,E1 -15413.776,E2 -15413.776} C_VEL
LIN {X 0,Y 327.157,Z 300.646,A -85,B 0,C 180,E1 -15416.128,E2 -15416.128} C_VEL
LIN {X 0,Y 325.353,Z 291.281,A -85,B 0,C 180,E1 -15418.623,E2 -15418.623} C_VEL
LIN {X 0,Y 324.067,Z 288.357,A -85,B 0,C 180,E1 -15419.497,E2 -15419.497} C_VEL
LIN {X 0,Y 320.197,Z 284.34,A -85,B 0,C 180,E1 -15420.954,E2 -15420.954} C_VEL
LIN {X 0,Y 316.916,Z 281.261,A -85,B 0,C 180,E1 -15422.147,E2 -15422.147} C_VEL
LIN {X 0,Y 315.155,Z 278.641,A -85,B 0,C 180,E1 -15423.066,E2 -15423.066} C_VEL
LIN {X 0,Y 314.81,Z 277.664,A -85,B 0,C 180,E1 -15423.375,E2 -15423.375} C_VEL
LIN {X 0,Y 312.546,Z 269.251,A -85,B 0,C 180,E1 -15426.072,E2 -15426.072} C_VEL
LIN {X 0,Y 312.504,Z 269.176,A -85,B 0,C 180,E1 -15430.124,E2 -15430.124} C_VEL
LIN {X 0,Y 312.458,Z 269.181,A -85,B 0,C 180,E1 -15433.964,E2 -15433.964} C_VEL
LIN {X 0,Y 312.483,Z 269.185,A -85,B 0,C 180,E1 -15437.918,E2 -15437.918} C_VEL
LIN {X 0,Y 312.533,Z 269.173,A -85,B 0,C 180,E1 -15441.91,E2 -15441.91} C_VEL
LIN {X 0,Y 312.504,Z 269.154,A -85,B 0,C 180,E1 -15445.789,E2 -15445.789} C_VEL
LIN {X 0,Y 312.521,Z 269.176,A -85,B 0,C 180,E1 -15448.853,E2 -15448.853} C_VEL
LIN {X 0,Y 312.572,Z 269.165,A -85,B 0,C 180,E1 -15451.824,E2 -15451.824} C_VEL
LIN {X 0,Y 312.582,Z 269.17,A -85,B 0,C 180,E1 -15454.71,E2 -15454.71} C_VEL
LIN {X 0,Y 312.583,Z 269.173,A -85,B 0,C 180,E1 -15457.528,E2 -15457.528} C_VEL
LIN {X 0,Y 312.634,Z 269.164,A -85,B 0,C 180,E1 -15461.656,E2 -15461.656} C_VEL
LIN {X 0,Y 312.689,Z 269.151,A -85,B 0,C 180,E1 -15465.685,E2 -15465.685} C_VEL
LIN {X 0,Y 312.693,Z 269.149,A -85,B 0,C 180,E1 -15469.641,E2 -15469.641} C_VEL
LIN {X 0,Y 312.848,Z 269.139,A -85,B 0,C 180,E1 -15472.253,E2 -15472.253} C_VEL
LIN {X 0,Y 312.71,Z 269.145,A -85,B 0,C 180,E1 -15474.842,E2 -15474.842} C_VEL
LIN {X 0,Y 312.985,Z 269.121,A -85,B 0,C 180,E1 -15478.713,E2 -15478.713} C_VEL
LIN {X 0,Y 312.985,Z 269.113,A -85,B 0,C 180,E1 -15481.286,E2 -15481.286} C_VEL
LIN {X 0,Y 312.712,Z 269.147,A -85,B 0,C 180,E1 -15485.157,E2 -15485.157} C_VEL
LIN {X 0,Y 312.866,Z 269.134,A -85,B 0,C 180,E1 -15487.745,E2 -15487.745} C_VEL
LIN {X 0,Y 312.663,Z 269.152,A -85,B 0,C 180,E1 -15491.671,E2 -15491.671} C_VEL
LIN {X 0,Y 312.694,Z 269.153,A -85,B 0,C 180,E1 -15494.887,E2 -15494.887} C_VEL
LIN {X 0,Y 312.625,Z 269.166,A -85,B 0,C 180,E1 -15499.236,E2 -15499.236} C_VEL
LIN {X 0,Y 312.54,Z 269.178,A -85,B 0,C 180,E1 -15502.789,E2 -15502.789} C_VEL
LIN {X 0,Y 312.598,Z 269.168,A -85,B 0,C 180,E1 -15505.936,E2 -15505.936} C_VEL
LIN {X 0,Y 312.54,Z 269.151,A -85,B 0,C 180,E1 -15509.65,E2 -15509.65} C_VEL
LIN {X 0,Y 312.515,Z 269.184,A -85,B 0,C 180,E1 -15513.689,E2 -15513.689} C_VEL
LIN {X 0,Y 312.521,Z 269.159,A -85,B 0,C 180,E1 -15517.385,E2 -15517.385} C_VEL
LIN {X 0,Y 312.485,Z 269.181,A -85,B 0,C 180,E1 -15520.71,E2 -15520.71} C_VEL
LIN {X 0,Y 312.469,Z 269.189,A -85,B 0,C 180,E1 -15524.206,E2 -15524.206} C_VEL
LIN {X 0,Y 312.482,Z 269.13,A -85,B 0,C 180,E1 -15527.919,E2 -15527.919} C_VEL
LIN {X 0,Y 312.529,Z 269.182,A -85,B 0,C 180,E1 -15532.037,E2 -15532.037} C_VEL
LIN {X 0,Y 312.559,Z 269.47,A -85,B 0,C 180,E1 -15532.361,E2 -15532.361} C_VEL
LIN {X 0,Y 315.556,Z 280.077,A -85,B 0,C 180,E1 -15535.493,E2 -15535.493} C_VEL
LIN {X 0,Y 318.519,Z 291.922,A -85,B 0,C 180,E1 -15538.753,E2 -15538.753} C_VEL
LIN {X 0,Y 320.411,Z 300.048,A -85,B 0,C 180,E1 -15540.796,E2 -15540.796} C_VEL
LIN {X 0,Y 323.532,Z 307.839,A -85,B 0,C 180,E1 -15541.302,E2 -15541.302} C_VEL
LIN {X 0,Y 327.011,Z 332.393,A -85,B 0,C 180,E1 -15542.216,E2 -15542.216} C_VEL
LIN {X 0,Y 324.24,Z 431.045,A -85,B 0,C 180,E1 -15544.482,E2 -15544.482} C_VEL
LIN {X 0,Y 323.302,Z 445.394,A -85,B 0,C 180,E1 -15545.049,E2 -15545.049} C_VEL
LIN {X 0,Y 322.149,Z 459.179,A -85,B 0,C 180,E1 -15545.855,E2 -15545.855} C_VEL
LIN {X 0,Y 320.861,Z 471.117,A -85,B 0,C 180,E1 -15546.78,E2 -15546.78} C_VEL
LIN {X 0,Y 319.381,Z 483.743,A -85,B 0,C 180,E1 -15548.033,E2 -15548.033} C_VEL
LIN {X 0,Y 317.664,Z 495.205,A -85,B 0,C 180,E1 -15549.439,E2 -15549.439} C_VEL
LIN {X 0,Y 316.221,Z 504.705,A -85,B 0,C 180,E1 -15550.864,E2 -15550.864} C_VEL
LIN {X 0,Y 314.623,Z 515.267,A -85,B 0,C 180,E1 -15552.784,E2 -15552.784} C_VEL
LIN {X 0,Y 313.4,Z 524.348,A -85,B 0,C 180,E1 -15554.836,E2 -15554.836} C_VEL
LIN {X 0,Y 312.351,Z 532.122,A -85,B 0,C 180,E1 -15556.997,E2 -15556.997} C_VEL
LIN {X 0,Y 311.529,Z 537.849,A -85,B 0,C 180,E1 -15558.945,E2 -15558.945} C_VEL
LIN {X 0,Y 311.121,Z 542.512,A -85,B 0,C 180,E1 -15560.902,E2 -15560.902} C_VEL
LIN {X 0,Y 310.83,Z 546.157,A -85,B 0,C 180,E1 -15562.857,E2 -15562.857} C_VEL
LIN {X 0,Y 310.683,Z 548.93,A -85,B 0,C 180,E1 -15564.809,E2 -15564.809} C_VEL
LIN {X 0,Y 310.674,Z 551.307,A -85,B 0,C 180,E1 -15567.407,E2 -15567.407} C_VEL
LIN {X 0,Y 310.69,Z 552.241,A -85,B 0,C 180,E1 -15570,E2 -15570} C_VEL
LIN {X 0,Y 310.673,Z 551.745,A -85,B 0,C 180,E1 -15572.593,E2 -15572.593} C_VEL
LIN {X 0,Y 310.688,Z 550.963,A -85,B 0,C 180,E1 -15573.891,E2 -15573.891} C_VEL
LIN {X 0,Y 310.809,Z 548.284,A -85,B 0,C 180,E1 -15576.492,E2 -15576.492} C_VEL
LIN {X 0,Y 311.149,Z 544.063,A -85,B 0,C 180,E1 -15579.097,E2 -15579.097} C_VEL
LIN {X 0,Y 311.635,Z 539.857,A -85,B 0,C 180,E1 -15581.051,E2 -15581.051} C_VEL
LIN {X 0,Y 312.622,Z 533.625,A -85,B 0,C 180,E1 -15583.322,E2 -15583.322} C_VEL
LIN {X 0,Y 313.796,Z 525.796,A -85,B 0,C 180,E1 -15585.59,E2 -15585.59} C_VEL
LIN {X 0,Y 315.161,Z 517.586,A -85,B 0,C 180,E1 -15587.52,E2 -15587.52} C_VEL
LIN {X 0,Y 316.9,Z 507.646,A -85,B 0,C 180,E1 -15589.43,E2 -15589.43} C_VEL
LIN {X 0,Y 318.79,Z 496.554,A -85,B 0,C 180,E1 -15591.161,E2 -15591.161} C_VEL
LIN {X 0,Y 320.537,Z 485.641,A -85,B 0,C 180,E1 -15592.543,E2 -15592.543} C_VEL
LIN {X 0,Y 322.176,Z 473.382,A -85,B 0,C 180,E1 -15593.8,E2 -15593.8} C_VEL
LIN {X 0,Y 323.773,Z 459.866,A -85,B 0,C 180,E1 -15594.87,E2 -15594.87} C_VEL
LIN {X 0,Y 325.148,Z 445.658,A -85,B 0,C 180,E1 -15595.699,E2 -15595.699} C_VEL
LIN {X 0,Y 326.14,Z 431.536,A -85,B 0,C 180,E1 -15596.259,E2 -15596.259} C_VEL
LIN {X 0,Y 329.075,Z 334.469,A -85,B 0,C 180,E1 -15598.491,E2 -15598.491} C_VEL
LIN {X 0,Y 328.751,Z 330.12,A -85,B 0,C 180,E1 -15598.632,E2 -15598.632} C_VEL
LIN {X 0,Y 325.649,Z 311.027,A -85,B 0,C 180,E1 -15599.417,E2 -15599.417} C_VEL
LIN {X 0,Y 320.849,Z 300,A -85,B 0,C 180,E1 -15600.217,E2 -15600.217} C_VEL
LIN {X 0,Y 317.795,Z 287.627,A -85,B 0,C 180,E1 -15603.564,E2 -15603.564} C_VEL
LIN {X 0,Y 314.981,Z 277.497,A -85,B 0,C 180,E1 -15606.559,E2 -15606.559} C_VEL
LIN {X 0,Y 312.558,Z 269.247,A -85,B 0,C 180,E1 -15609.22,E2 -15609.22} C_VEL
LIN {X 0,Y 312.546,Z 269.18,A -85,B 0,C 180,E1 -15612.421,E2 -15612.421} C_VEL
LIN {X 0,Y 312.516,Z 269.18,A -85,B 0,C 180,E1 -15616.023,E2 -15616.023} C_VEL
LIN {X 0,Y 312.5,Z 269.171,A -85,B 0,C 180,E1 -15619.874,E2 -15619.874} C_VEL
LIN {X 0,Y 312.533,Z 269.166,A -85,B 0,C 180,E1 -15622.616,E2 -15622.616} C_VEL
LIN {X 0,Y 312.515,Z 269.18,A -85,B 0,C 180,E1 -15626.311,E2 -15626.311} C_VEL
LIN {X 0,Y 312.541,Z 269.147,A -85,B 0,C 180,E1 -15630.35,E2 -15630.35} C_VEL
LIN {X 0,Y 312.598,Z 269.171,A -85,B 0,C 180,E1 -15634.064,E2 -15634.064} C_VEL
LIN {X 0,Y 312.583,Z 269.174,A -85,B 0,C 180,E1 -15637.529,E2 -15637.529} C_VEL
LIN {X 0,Y 312.633,Z 269.169,A -85,B 0,C 180,E1 -15641.656,E2 -15641.656} C_VEL
LIN {X 0,Y 312.689,Z 269.16,A -85,B 0,C 180,E1 -15645.686,E2 -15645.686} C_VEL
LIN {X 0,Y 312.696,Z 269.155,A -85,B 0,C 180,E1 -15649.642,E2 -15649.642} C_VEL
LIN {X 0,Y 312.861,Z 269.126,A -85,B 0,C 180,E1 -15652.254,E2 -15652.254} C_VEL
LIN {X 0,Y 312.712,Z 269.156,A -85,B 0,C 180,E1 -15654.843,E2 -15654.843} C_VEL
LIN {X 0,Y 312.986,Z 269.118,A -85,B 0,C 180,E1 -15658.714,E2 -15658.714} C_VEL
LIN {X 0,Y 312.986,Z 269.116,A -85,B 0,C 180,E1 -15661.287,E2 -15661.287} C_VEL
LIN {X 0,Y 312.713,Z 269.158,A -85,B 0,C 180,E1 -15665.158,E2 -15665.158} C_VEL
LIN {X 0,Y 312.867,Z 269.13,A -85,B 0,C 180,E1 -15667.746,E2 -15667.746} C_VEL
LIN {X 0,Y 312.665,Z 269.153,A -85,B 0,C 180,E1 -15671.672,E2 -15671.672} C_VEL
LIN {X 0,Y 312.696,Z 269.154,A -85,B 0,C 180,E1 -15674.888,E2 -15674.888} C_VEL
LIN {X 0,Y 312.627,Z 269.161,A -85,B 0,C 180,E1 -15679.237,E2 -15679.237} C_VEL
LIN {X 0,Y 312.543,Z 269.177,A -85,B 0,C 180,E1 -15682.79,E2 -15682.79} C_VEL
LIN {X 0,Y 312.6,Z 269.172,A -85,B 0,C 180,E1 -15685.936,E2 -15685.936} C_VEL
LIN {X 0,Y 312.535,Z 269.152,A -85,B 0,C 180,E1 -15689.652,E2 -15689.652} C_VEL
LIN {X 0,Y 312.518,Z 269.169,A -85,B 0,C 180,E1 -15693.69,E2 -15693.69} C_VEL
LIN {X 0,Y 312.537,Z 269.181,A -85,B 0,C 180,E1 -15697.384,E2 -15697.384} C_VEL
LIN {X 0,Y 312.489,Z 269.168,A -85,B 0,C 180,E1 -15700.71,E2 -15700.71} C_VEL
LIN {X 0,Y 312.451,Z 269.176,A -85,B 0,C 180,E1 -15704.211,E2 -15704.211} C_VEL
LIN {X 0,Y 312.498,Z 269.201,A -85,B 0,C 180,E1 -15708.365,E2 -15708.365} C_VEL
LIN {X 0,Y 312.58,Z 269.656,A -85,B 0,C 180,E1 -15708.71,E2 -15708.71} C_VEL
LIN {X 0,Y 315.282,Z 278.927,A -85,B 0,C 180,E1 -15711.792,E2 -15711.792} C_VEL
LIN {X 0,Y 317.924,Z 289.032,A -85,B 0,C 180,E1 -15714.918,E2 -15714.918} C_VEL
LIN {X 0,Y 320.802,Z 302.218,A -85,B 0,C 180,E1 -15718.694,E2 -15718.694} C_VEL
LIN {X 0,Y 321.259,Z 306.328,A -85,B 0,C 180,E1 -15719.791,E2 -15719.791} C_VEL
LIN {X 0,Y 320.52,Z 310.859,A -85,B 0,C 180,E1 -15720.813,E2 -15720.813} C_VEL
LIN {X 0,Y 325.261,Z 334.992,A -85,B 0,C 180,E1 -15721.886,E2 -15721.886} C_VEL
LIN {X 0,Y 328.203,Z 352.292,A -85,B 0,C 180,E1 -15722.563,E2 -15722.563} C_VEL
LIN {X 0,Y 326.338,Z 426.176,A -85,B 0,C 180,E1 -15724.102,E2 -15724.102} C_VEL
LIN {X 0,Y 325.474,Z 439.311,A -85,B 0,C 180,E1 -15724.586,E2 -15724.586} C_VEL
LIN {X 0,Y 324.391,Z 452.581,A -85,B 0,C 180,E1 -15725.352,E2 -15725.352} C_VEL
LIN {X 0,Y 323.115,Z 464.222,A -85,B 0,C 180,E1 -15726.265,E2 -15726.265} C_VEL
LIN {X 0,Y 321.604,Z 475.005,A -85,B 0,C 180,E1 -15727.347,E2 -15727.347} C_VEL
LIN {X 0,Y 319.771,Z 486.017,A -85,B 0,C 180,E1 -15728.738,E2 -15728.738} C_VEL
LIN {X 0,Y 317.955,Z 495.872,A -85,B 0,C 180,E1 -15730.301,E2 -15730.301} C_VEL
LIN {X 0,Y 316.084,Z 505.453,A -85,B 0,C 180,E1 -15732.198,E2 -15732.198} C_VEL
LIN {X 0,Y 314.649,Z 512.829,A -85,B 0,C 180,E1 -15734.022,E2 -15734.022} C_VEL
LIN {X 0,Y 313.649,Z 518.444,A -85,B 0,C 180,E1 -15735.731,E2 -15735.731} C_VEL
LIN {X 0,Y 312.5,Z 523.637,A -85,B 0,C 180,E1 -15737.664,E2 -15737.664} C_VEL
LIN {X 0,Y 311.82,Z 527.723,A -85,B 0,C 180,E1 -15739.612,E2 -15739.612} C_VEL
LIN {X 0,Y 311.458,Z 529.907,A -85,B 0,C 180,E1 -15740.912,E2 -15740.912} C_VEL
LIN {X 0,Y 311.186,Z 531.675,A -85,B 0,C 180,E1 -15742.212,E2 -15742.212} C_VEL
LIN {X 0,Y 310.825,Z 533.987,A -85,B 0,C 180,E1 -15744.811,E2 -15744.811} C_VEL
LIN {X 0,Y 310.803,Z 534.595,A -85,B 0,C 180,E1 -15746.11,E2 -15746.11} C_VEL
LIN {X 0,Y 310.686,Z 534.748,A -85,B 0,C 180,E1 -15748.704,E2 -15748.704} C_VEL
LIN {X 0,Y 310.768,Z 533.401,A -85,B 0,C 180,E1 -15751.296,E2 -15751.296} C_VEL
LIN {X 0,Y 311.149,Z 530.576,A -85,B 0,C 180,E1 -15753.885,E2 -15753.885} C_VEL
LIN {X 0,Y 311.626,Z 527.397,A -85,B 0,C 180,E1 -15755.825,E2 -15755.825} C_VEL
LIN {X 0,Y 312.315,Z 522.53,A -85,B 0,C 180,E1 -15758.052,E2 -15758.052} C_VEL
LIN {X 0,Y 313.335,Z 515.965,A -85,B 0,C 180,E1 -15760.337,E2 -15760.337} C_VEL
LIN {X 0,Y 314.57,Z 508.938,A -85,B 0,C 180,E1 -15762.254,E2 -15762.254} C_VEL
LIN {X 0,Y 316.096,Z 500.259,A -85,B 0,C 180,E1 -15764.156,E2 -15764.156} C_VEL
LIN {X 0,Y 317.491,Z 491.42,A -85,B 0,C 180,E1 -15765.733,E2 -15765.733} C_VEL
LIN {X 0,Y 319.024,Z 481.747,A -85,B 0,C 180,E1 -15767.136,E2 -15767.136} C_VEL
LIN {X 0,Y 320.397,Z 471.213,A -85,B 0,C 180,E1 -15768.38,E2 -15768.38} C_VEL
LIN {X 0,Y 321.864,Z 459.573,A -85,B 0,C 180,E1 -15769.45,E2 -15769.45} C_VEL
LIN {X 0,Y 323.062,Z 447.581,A -85,B 0,C 180,E1 -15770.286,E2 -15770.286} C_VEL
LIN {X 0,Y 323.903,Z 434.575,A -85,B 0,C 180,E1 -15770.94,E2 -15770.94} C_VEL
LIN {X 0,Y 324.529,Z 420.653,A -85,B 0,C 180,E1 -15771.363,E2 -15771.363} C_VEL
LIN {X 0,Y 325.96,Z 349.949,A -85,B 0,C 180,E1 -15772.836,E2 -15772.836} C_VEL
LIN {X 0,Y 320.48,Z 317.679,A -85,B 0,C 180,E1 -15774.045,E2 -15774.045} C_VEL
LIN {X 0,Y 319.226,Z 310.973,A -85,B 0,C 180,E1 -15774.349,E2 -15774.349} C_VEL
LIN {X 0,Y 320.304,Z 302.179,A -85,B 0,C 180,E1 -15776.379,E2 -15776.379} C_VEL
LIN {X 0,Y 317.928,Z 290.109,A -85,B 0,C 180,E1 -15779.694,E2 -15779.694} C_VEL
LIN {X 0,Y 314.81,Z 277.664,A -85,B 0,C 180,E1 -15783.375,E2 -15783.375} C_VEL
LIN {X 0,Y 313.625,Z 275.965,A -85,B 0,C 180,E1 -15783.992,E2 -15783.992} C_VEL
LIN {X 0,Y 306.62,Z 272.139,A -85,B 0,C 180,E1 -15786.008,E2 -15786.008} C_VEL
LIN {X 0,Y 305.574,Z 270.458,A -85,B 0,C 180,E1 -15786.661,E2 -15786.661} C_VEL
LIN {X 0,Y 305.477,Z 270.052,A -85,B 0,C 180,E1 -15787.151,E2 -15787.151} C_VEL
LIN {X 0,Y 305.455,Z 270.05,A -85,B 0,C 180,E1 -15790.599,E2 -15790.599} C_VEL
LIN {X 0,Y 305.425,Z 270.061,A -85,B 0,C 180,E1 -15793.654,E2 -15793.654} C_VEL
LIN {X 0,Y 305.454,Z 270.064,A -85,B 0,C 180,E1 -15797.413,E2 -15797.413} C_VEL
LIN {X 0,Y 305.493,Z 270.043,A -85,B 0,C 180,E1 -15801.599,E2 -15801.599} C_VEL
LIN {X 0,Y 305.46,Z 270.041,A -85,B 0,C 180,E1 -15804.886,E2 -15804.886} C_VEL
LIN {X 0,Y 305.45,Z 270.053,A -85,B 0,C 180,E1 -15808.354,E2 -15808.354} C_VEL
LIN {X 0,Y 305.518,Z 270.046,A -85,B 0,C 180,E1 -15811.113,E2 -15811.113} C_VEL
LIN {X 0,Y 305.569,Z 270.047,A -85,B 0,C 180,E1 -15814.087,E2 -15814.087} C_VEL
LIN {X 0,Y 305.496,Z 270.057,A -85,B 0,C 180,E1 -15818.402,E2 -15818.402} C_VEL
LIN {X 0,Y 305.586,Z 270.039,A -85,B 0,C 180,E1 -15821.217,E2 -15821.217} C_VEL
LIN {X 0,Y 305.644,Z 270.026,A -85,B 0,C 180,E1 -15825.348,E2 -15825.348} C_VEL
LIN {X 0,Y 305.63,Z 270.029,A -85,B 0,C 180,E1 -15829.399,E2 -15829.399} C_VEL
LIN {X 0,Y 305.792,Z 270.017,A -85,B 0,C 180,E1 -15832.073,E2 -15832.073} C_VEL
LIN {X 0,Y 305.681,Z 270.021,A -85,B 0,C 180,E1 -15834.723,E2 -15834.723} C_VEL
LIN {X 0,Y 305.952,Z 269.998,A -85,B 0,C 180,E1 -15838.683,E2 -15838.683} C_VEL
LIN {X 0,Y 305.952,Z 269.989,A -85,B 0,C 180,E1 -15841.316,E2 -15841.316} C_VEL
LIN {X 0,Y 305.846,Z 270.002,A -85,B 0,C 180,E1 -15846.597,E2 -15846.597} C_VEL
LIN {X 0,Y 305.73,Z 270.024,A -85,B 0,C 180,E1 -15849.259,E2 -15849.259} C_VEL
LIN {X 0,Y 305.583,Z 270.044,A -85,B 0,C 180,E1 -15853.296,E2 -15853.296} C_VEL
LIN {X 0,Y 305.588,Z 270.034,A -85,B 0,C 180,E1 -15856.02,E2 -15856.02} C_VEL
LIN {X 0,Y 305.571,Z 270.044,A -85,B 0,C 180,E1 -15859.445,E2 -15859.445} C_VEL
LIN {X 0,Y 305.485,Z 270.057,A -85,B 0,C 180,E1 -15863.041,E2 -15863.041} C_VEL
LIN {X 0,Y 305.543,Z 270.05,A -85,B 0,C 180,E1 -15866.227,E2 -15866.227} C_VEL
LIN {X 0,Y 305.491,Z 270.035,A -85,B 0,C 180,E1 -15869.05,E2 -15869.05} C_VEL
LIN {X 0,Y 305.439,Z 270.045,A -85,B 0,C 180,E1 -15871.952,E2 -15871.952} C_VEL
LIN {X 0,Y 305.458,Z 270.053,A -85,B 0,C 180,E1 -15875.113,E2 -15875.113} C_VEL
LIN {X 0,Y 305.445,Z 270.054,A -85,B 0,C 180,E1 -15878.529,E2 -15878.529} C_VEL
LIN {X 0,Y 305.455,Z 270.045,A -85,B 0,C 180,E1 -15882.587,E2 -15882.587} C_VEL
LIN {X 0,Y 305.439,Z 270.025,A -85,B 0,C 180,E1 -15886.348,E2 -15886.348} C_VEL
LIN {X 0,Y 305.454,Z 270.021,A -85,B 0,C 180,E1 -15889.893,E2 -15889.893} C_VEL
LIN {X 0,Y 305.477,Z 270.205,A -85,B 0,C 180,E1 -15891.556,E2 -15891.556} C_VEL
LIN {X 0,Y 308.316,Z 280.011,A -85,B 0,C 180,E1 -15894.578,E2 -15894.578} C_VEL
LIN {X 0,Y 311.345,Z 291.862,A -85,B 0,C 180,E1 -15897.964,E2 -15897.964} C_VEL
LIN {X 0,Y 313.223,Z 300.081,A -85,B 0,C 180,E1 -15900.117,E2 -15900.117} C_VEL
LIN {X 0,Y 317.472,Z 310.662,A -85,B 0,C 180,E1 -15900.829,E2 -15900.829} C_VEL
LIN {X 0,Y 320.609,Z 333.574,A -85,B 0,C 180,E1 -15901.697,E2 -15901.697} C_VEL
LIN {X 0,Y 317.762,Z 430.793,A -85,B 0,C 180,E1 -15903.968,E2 -15903.968} C_VEL
LIN {X 0,Y 316.797,Z 445.212,A -85,B 0,C 180,E1 -15904.544,E2 -15904.544} C_VEL
LIN {X 0,Y 315.744,Z 457.326,A -85,B 0,C 180,E1 -15905.246,E2 -15905.246} C_VEL
LIN {X 0,Y 314.311,Z 470.532,A -85,B 0,C 180,E1 -15906.267,E2 -15906.267} C_VEL
